MOVL C04706 V=8.0
MOVL C04707 V=8.0
MOVL C04708 V=8.0
MOVL C04709 V=8.0
MOVL C04710 V=8.0
MOVL C04711 V=8.0
MOVL C04712 V=8.0
MOVL C04713 V=8.0
MOVL C04714 V=8.0
MOVL C04715 V=8.0
MOVL C04716 V=8.0
MOVL C04717 V=8.0
MOVL C04718 V=8.0
MOVL C04719 V=8.0
MOVL C04720 V=8.0
MOVL C04721 V=8.0
MOVL C04722 V=8.0
MOVJ C04723 VJ=0.78
MOVJ C04724 VJ=0.78
MOVL C04725 V=11.7
TIMER T=2.00
MOVL C04726 V=11.7
MOVJ C04727 VJ=0.78
MOVJ C04728 VJ=0.78
MOVL C04729 V=8.0
MOVL C04730 V=8.0
MOVJ C04731 VJ=0.78
MOVL C04732 V=8.0
MOVL C04733 V=8.0
MOVL C04734 V=8.0
MOVL C04735 V=8.0
MOVL C04736 V=8.0
MOVL C04737 V=8.0
MOVL C04738 V=8.0
MOVL C04739 V=8.0
MOVL C04740 V=8.0
MOVL C04741 V=8.0
MOVL C04742 V=8.0
MOVL C04743 V=8.0
MOVL C04744 V=8.0
MOVL C04745 V=8.0
MOVL C04746 V=8.0
MOVL C04747 V=8.0
MOVL C04748 V=8.0
MOVL C04749 V=8.0
MOVL C04750 V=8.0
MOVL C04751 V=8.0
MOVL C04752 V=8.0
MOVL C04753 V=8.0
MOVL C04754 V=8.0
MOVL C04755 V=8.0
MOVL C04756 V=8.0
MOVL C04757 V=8.0
MOVL C04758 V=8.0
MOVL C04759 V=8.0
MOVL C04760 V=8.0
MOVL C04761 V=8.0
MOVL C04762 V=8.0
MOVL C04763 V=8.0
MOVL C04764 V=8.0
MOVL C04765 V=8.0
MOVL C04766 V=8.0
MOVL C04767 V=8.0
MOVL C04768 V=8.0
MOVL C04769 V=8.0
MOVL C04770 V=8.0
MOVL C04771 V=8.0
MOVL C04772 V=8.0
MOVL C04773 V=8.0
MOVL C04774 V=8.0
MOVL C04775 V=8.0
MOVL C04776 V=8.0
MOVL C04777 V=8.0
MOVL C04778 V=8.0
MOVL C04779 V=8.0
MOVL C04780 V=8.0
MOVL C04781 V=8.0
MOVL C04782 V=8.0
MOVL C04783 V=8.0
MOVL C04784 V=8.0
MOVL C04785 V=8.0
MOVL C04786 V=8.0
MOVL C04787 V=8.0
MOVL C04788 V=8.0
MOVL C04789 V=8.0
MOVL C04790 V=8.0
MOVL C04791 V=8.0
MOVL C04792 V=8.0
MOVL C04793 V=8.0
MOVJ C04794 VJ=0.78
MOVL C04795 V=8.0
MOVL C04796 V=8.0
MOVL C04797 V=8.0
MOVL C04798 V=8.0
MOVL C04799 V=8.0
MOVL C04800 V=8.0
MOVL C04801 V=8.0
MOVL C04802 V=8.0
MOVL C04803 V=8.0
MOVL C04804 V=8.0
MOVL C04805 V=8.0
MOVL C04806 V=8.0
MOVL C04807 V=8.0
MOVL C04808 V=8.0
MOVL C04809 V=8.0
MOVL C04810 V=8.0
MOVL C04811 V=8.0
MOVL C04812 V=8.0
MOVL C04813 V=8.0
MOVL C04814 V=8.0
MOVL C04815 V=8.0
MOVL C04816 V=8.0
MOVL C04817 V=8.0
MOVL C04818 V=8.0
MOVL C04819 V=8.0
MOVL C04820 V=8.0
MOVL C04821 V=8.0
MOVL C04822 V=8.0
MOVL C04823 V=8.0
MOVL C04824 V=8.0
MOVL C04825 V=8.0
MOVL C04826 V=8.0
MOVL C04827 V=8.0
MOVL C04828 V=8.0
MOVL C04829 V=8.0
MOVL C04830 V=8.0
MOVL C04831 V=8.0
MOVL C04832 V=8.0
MOVL C04833 V=8.0
MOVL C04834 V=8.0
MOVL C04835 V=8.0
MOVL C04836 V=8.0
MOVL C04837 V=8.0
MOVL C04838 V=8.0
MOVL C04839 V=8.0
MOVL C04840 V=8.0
MOVL C04841 V=8.0
MOVL C04842 V=8.0
MOVL C04843 V=8.0
MOVL C04844 V=8.0
MOVL C04845 V=8.0
MOVL C04846 V=8.0
MOVL C04847 V=8.0
MOVL C04848 V=8.0
MOVL C04849 V=8.0
MOVL C04850 V=8.0
MOVL C04851 V=8.0
MOVL C04852 V=8.0
MOVL C04853 V=8.0
MOVL C04854 V=8.0
MOVL C04855 V=8.0
MOVL C04856 V=8.0
MOVJ C04857 VJ=0.78
MOVL C04858 V=8.0
MOVL C04859 V=8.0
MOVL C04860 V=8.0
MOVL C04861 V=8.0
MOVL C04862 V=8.0
MOVL C04863 V=8.0
MOVL C04864 V=8.0
MOVL C04865 V=8.0
MOVL C04866 V=8.0
MOVL C04867 V=8.0
MOVL C04868 V=8.0
MOVL C04869 V=8.0
MOVL C04870 V=8.0
MOVL C04871 V=8.0
MOVL C04872 V=8.0
MOVL C04873 V=8.0
MOVL C04874 V=8.0
MOVL C04875 V=8.0
MOVL C04876 V=8.0
MOVL C04877 V=8.0
MOVL C04878 V=8.0
MOVL C04879 V=8.0
MOVL C04880 V=8.0
MOVL C04881 V=8.0
MOVL C04882 V=8.0
MOVL C04883 V=8.0
MOVL C04884 V=8.0
MOVL C04885 V=8.0
MOVL C04886 V=8.0
MOVL C04887 V=8.0
MOVL C04888 V=8.0
MOVL C04889 V=8.0
MOVL C04890 V=8.0
MOVL C04891 V=8.0
MOVL C04892 V=8.0
MOVL C04893 V=8.0
MOVL C04894 V=8.0
MOVL C04895 V=8.0
MOVL C04896 V=8.0
MOVL C04897 V=8.0
MOVL C04898 V=8.0
MOVJ C04899 VJ=0.78
MOVJ C04900 VJ=0.78
MOVL C04901 V=11.7
TIMER T=2.00
MOVL C04902 V=11.7
MOVJ C04903 VJ=0.78
MOVJ C04904 VJ=0.78
MOVL C04905 V=8.0
MOVL C04906 V=8.0
MOVL C04907 V=8.0
MOVL C04908 V=8.0
MOVL C04909 V=8.0
MOVL C04910 V=8.0
MOVL C04911 V=8.0
MOVL C04912 V=8.0
MOVL C04913 V=8.0
MOVL C04914 V=8.0
MOVL C04915 V=8.0
MOVL C04916 V=8.0
MOVL C04917 V=8.0
MOVL C04918 V=8.0
MOVL C04919 V=8.0
MOVL C04920 V=8.0
MOVL C04921 V=8.0
MOVL C04922 V=8.0
MOVL C04923 V=8.0
MOVL C04924 V=8.0
MOVL C04925 V=8.0
MOVL C04926 V=8.0
MOVJ C04927 VJ=0.78
MOVL C04928 V=8.0
MOVL C04929 V=8.0
MOVL C04930 V=8.0
MOVL C04931 V=8.0
MOVL C04932 V=8.0
MOVL C04933 V=8.0
MOVL C04934 V=8.0
MOVL C04935 V=8.0
MOVL C04936 V=8.0
MOVL C04937 V=8.0
MOVL C04938 V=8.0
MOVL C04939 V=8.0
MOVL C04940 V=8.0
MOVL C04941 V=8.0
MOVL C04942 V=8.0
MOVL C04943 V=8.0
MOVL C04944 V=8.0
MOVL C04945 V=8.0
MOVL C04946 V=8.0
MOVL C04947 V=8.0
MOVL C04948 V=8.0
MOVL C04949 V=8.0
MOVL C04950 V=8.0
MOVL C04951 V=8.0
MOVL C04952 V=8.0
MOVL C04953 V=8.0
MOVL C04954 V=8.0
MOVL C04955 V=8.0
MOVL C04956 V=8.0
MOVL C04957 V=8.0
MOVL C04958 V=8.0
MOVL C04959 V=8.0
MOVL C04960 V=8.0
MOVL C04961 V=8.0
MOVL C04962 V=8.0
MOVL C04963 V=8.0
MOVL C04964 V=8.0
MOVL C04965 V=8.0
MOVL C04966 V=8.0
MOVL C04967 V=8.0
MOVL C04968 V=8.0
MOVL C04969 V=8.0
MOVL C04970 V=8.0
MOVL C04971 V=8.0
MOVL C04972 V=8.0
MOVL C04973 V=8.0
MOVL C04974 V=8.0
MOVL C04975 V=8.0
MOVL C04976 V=8.0
MOVL C04977 V=8.0
MOVL C04978 V=8.0
MOVL C04979 V=8.0
MOVL C04980 V=8.0
MOVL C04981 V=8.0
MOVL C04982 V=8.0
MOVL C04983 V=8.0
MOVL C04984 V=8.0
MOVL C04985 V=8.0
MOVL C04986 V=8.0
MOVL C04987 V=8.0
MOVL C04988 V=8.0
MOVL C04989 V=8.0
MOVJ C04990 VJ=0.78
MOVL C04991 V=8.0
MOVL C04992 V=8.0
MOVL C04993 V=8.0
MOVL C04994 V=8.0
MOVL C04995 V=8.0
MOVL C04996 V=8.0
MOVL C04997 V=8.0
MOVL C04998 V=8.0
MOVL C04999 V=8.0
MOVL C05000 V=8.0
MOVL C05001 V=8.0
MOVL C05002 V=8.0
MOVL C05003 V=8.0
MOVL C05004 V=8.0
MOVL C05005 V=8.0
MOVL C05006 V=8.0
MOVL C05007 V=8.0
MOVL C05008 V=8.0
MOVL C05009 V=8.0
MOVL C05010 V=8.0
MOVL C05011 V=8.0
MOVL C05012 V=8.0
MOVL C05013 V=8.0
MOVL C05014 V=8.0
MOVL C05015 V=8.0
MOVL C05016 V=8.0
MOVL C05017 V=8.0
MOVL C05018 V=8.0
MOVL C05019 V=8.0
MOVL C05020 V=8.0
MOVL C05021 V=8.0
MOVL C05022 V=8.0
MOVL C05023 V=8.0
MOVL C05024 V=8.0
MOVL C05025 V=8.0
MOVL C05026 V=8.0
MOVL C05027 V=8.0
MOVL C05028 V=8.0
MOVL C05029 V=8.0
MOVL C05030 V=8.0
MOVL C05031 V=8.0
MOVL C05032 V=8.0
MOVL C05033 V=8.0
MOVL C05034 V=8.0
MOVL C05035 V=8.0
MOVL C05036 V=8.0
MOVL C05037 V=8.0
MOVL C05038 V=8.0
MOVL C05039 V=8.0
MOVL C05040 V=8.0
MOVL C05041 V=8.0
MOVL C05042 V=8.0
MOVL C05043 V=8.0
MOVL C05044 V=8.0
MOVL C05045 V=8.0
MOVL C05046 V=8.0
MOVL C05047 V=8.0
MOVL C05048 V=8.0
MOVL C05049 V=8.0
MOVL C05050 V=8.0
MOVL C05051 V=8.0
MOVL C05052 V=8.0
MOVJ C05053 VJ=0.78
MOVL C05054 V=8.0
MOVL C05055 V=8.0
MOVL C05056 V=8.0
MOVL C05057 V=8.0
MOVL C05058 V=8.0
MOVL C05059 V=8.0
MOVL C05060 V=8.0
MOVL C05061 V=8.0
MOVL C05062 V=8.0
MOVL C05063 V=8.0
MOVL C05064 V=8.0
MOVL C05065 V=8.0
MOVL C05066 V=8.0
MOVL C05067 V=8.0
MOVL C05068 V=8.0
MOVL C05069 V=8.0
MOVL C05070 V=8.0
MOVL C05071 V=8.0
MOVL C05072 V=8.0
MOVL C05073 V=8.0
MOVL C05074 V=8.0
MOVJ C05075 VJ=0.78
MOVJ C05076 VJ=0.78
MOVL C05077 V=11.7
TIMER T=2.00
MOVL C05078 V=11.7
MOVJ C05079 VJ=0.78
MOVJ C05080 VJ=0.78
MOVL C05081 V=8.0
MOVL C05082 V=8.0
MOVL C05083 V=8.0
MOVL C05084 V=8.0
MOVL C05085 V=8.0
MOVL C05086 V=8.0
MOVL C05087 V=8.0
MOVL C05088 V=8.0
MOVL C05089 V=8.0
MOVL C05090 V=8.0
MOVL C05091 V=8.0
MOVL C05092 V=8.0
MOVL C05093 V=8.0
MOVL C05094 V=8.0
MOVL C05095 V=8.0
MOVL C05096 V=8.0
MOVL C05097 V=8.0
MOVL C05098 V=8.0
MOVL C05099 V=8.0
MOVL C05100 V=8.0
MOVL C05101 V=8.0
MOVL C05102 V=8.0
MOVL C05103 V=8.0
MOVL C05104 V=8.0
MOVL C05105 V=8.0
MOVL C05106 V=8.0
MOVL C05107 V=8.0
MOVL C05108 V=8.0
MOVL C05109 V=8.0
MOVL C05110 V=8.0
MOVL C05111 V=8.0
MOVL C05112 V=8.0
MOVL C05113 V=8.0
MOVL C05114 V=8.0
MOVL C05115 V=8.0
MOVL C05116 V=8.0
MOVL C05117 V=8.0
MOVL C05118 V=8.0
MOVL C05119 V=8.0
MOVL C05120 V=8.0
MOVL C05121 V=8.0
MOVL C05122 V=8.0
MOVJ C05123 VJ=0.78
MOVL C05124 V=8.0
MOVL C05125 V=8.0
MOVL C05126 V=8.0
MOVL C05127 V=8.0
MOVL C05128 V=8.0
MOVL C05129 V=8.0
MOVL C05130 V=8.0
MOVL C05131 V=8.0
MOVL C05132 V=8.0
MOVL C05133 V=8.0
MOVL C05134 V=8.0
MOVL C05135 V=8.0
MOVL C05136 V=8.0
MOVL C05137 V=8.0
MOVL C05138 V=8.0
MOVL C05139 V=8.0
MOVL C05140 V=8.0
MOVL C05141 V=8.0
MOVL C05142 V=8.0
MOVL C05143 V=8.0
MOVL C05144 V=8.0
MOVL C05145 V=8.0
MOVL C05146 V=8.0
MOVL C05147 V=8.0
MOVL C05148 V=8.0
MOVL C05149 V=8.0
MOVL C05150 V=8.0
MOVL C05151 V=8.0
MOVL C05152 V=8.0
MOVL C05153 V=8.0
MOVL C05154 V=8.0
MOVL C05155 V=8.0
MOVL C05156 V=8.0
MOVL C05157 V=8.0
MOVL C05158 V=8.0
MOVL C05159 V=8.0
MOVL C05160 V=8.0
MOVL C05161 V=8.0
MOVL C05162 V=8.0
MOVL C05163 V=8.0
MOVL C05164 V=8.0
MOVL C05165 V=8.0
MOVL C05166 V=8.0
MOVL C05167 V=8.0
MOVL C05168 V=8.0
MOVL C05169 V=8.0
MOVL C05170 V=8.0
MOVL C05171 V=8.0
MOVL C05172 V=8.0
MOVL C05173 V=8.0
MOVL C05174 V=8.0
MOVL C05175 V=8.0
MOVL C05176 V=8.0
MOVL C05177 V=8.0
MOVL C05178 V=8.0
MOVL C05179 V=8.0
MOVL C05180 V=8.0
MOVL C05181 V=8.0
MOVL C05182 V=8.0
MOVL C05183 V=8.0
MOVL C05184 V=8.0
MOVL C05185 V=8.0
MOVJ C05186 VJ=0.78
MOVL C05187 V=8.0
MOVL C05188 V=8.0
MOVL C05189 V=8.0
MOVL C05190 V=8.0
MOVL C05191 V=8.0
MOVL C05192 V=8.0
MOVL C05193 V=8.0
MOVL C05194 V=8.0
MOVL C05195 V=8.0
MOVL C05196 V=8.0
MOVL C05197 V=8.0
MOVL C05198 V=8.0
MOVL C05199 V=8.0
MOVL C05200 V=8.0
MOVL C05201 V=8.0
MOVL C05202 V=8.0
MOVL C05203 V=8.0
MOVL C05204 V=8.0
MOVL C05205 V=8.0
MOVL C05206 V=8.0
MOVL C05207 V=8.0
MOVL C05208 V=8.0
MOVL C05209 V=8.0
MOVL C05210 V=8.0
MOVL C05211 V=8.0
MOVL C05212 V=8.0
MOVL C05213 V=8.0
MOVL C05214 V=8.0
MOVL C05215 V=8.0
MOVL C05216 V=8.0
MOVL C05217 V=8.0
MOVL C05218 V=8.0
MOVL C05219 V=8.0
MOVL C05220 V=8.0
MOVL C05221 V=8.0
MOVL C05222 V=8.0
MOVL C05223 V=8.0
MOVL C05224 V=8.0
MOVL C05225 V=8.0
MOVL C05226 V=8.0
MOVL C05227 V=8.0
MOVL C05228 V=8.0
MOVL C05229 V=8.0
MOVL C05230 V=8.0
MOVL C05231 V=8.0
MOVL C05232 V=8.0
MOVL C05233 V=8.0
MOVL C05234 V=8.0
MOVL C05235 V=8.0
MOVL C05236 V=8.0
MOVL C05237 V=8.0
MOVL C05238 V=8.0
MOVL C05239 V=8.0
MOVL C05240 V=8.0
MOVL C05241 V=8.0
MOVL C05242 V=8.0
MOVL C05243 V=8.0
MOVL C05244 V=8.0
MOVL C05245 V=8.0
MOVL C05246 V=8.0
MOVL C05247 V=8.0
MOVJ C05248 VJ=0.78
MOVJ C05249 VJ=0.78
MOVL C05250 V=11.7
TIMER T=2.00
MOVL C05251 V=11.7
MOVJ C05252 VJ=0.78
MOVJ C05253 VJ=0.78
MOVL C05254 V=8.0
MOVL C05255 V=8.0
MOVJ C05256 VJ=0.78
MOVL C05257 V=8.0
MOVL C05258 V=8.0
MOVL C05259 V=8.0
MOVL C05260 V=8.0
MOVL C05261 V=8.0
MOVL C05262 V=8.0
MOVL C05263 V=8.0
MOVL C05264 V=8.0
MOVL C05265 V=8.0
MOVL C05266 V=8.0
MOVL C05267 V=8.0
MOVL C05268 V=8.0
MOVL C05269 V=8.0
MOVL C05270 V=8.0
MOVL C05271 V=8.0
MOVL C05272 V=8.0
MOVL C05273 V=8.0
MOVL C05274 V=8.0
MOVL C05275 V=8.0
MOVL C05276 V=8.0
MOVL C05277 V=8.0
MOVL C05278 V=8.0
MOVL C05279 V=8.0
MOVL C05280 V=8.0
MOVL C05281 V=8.0
MOVL C05282 V=8.0
MOVL C05283 V=8.0
MOVL C05284 V=8.0
MOVL C05285 V=8.0
MOVL C05286 V=8.0
MOVL C05287 V=8.0
MOVL C05288 V=8.0
MOVL C05289 V=8.0
MOVL C05290 V=8.0
MOVL C05291 V=8.0
MOVL C05292 V=8.0
MOVL C05293 V=8.0
MOVL C05294 V=8.0
MOVL C05295 V=8.0
MOVL C05296 V=8.0
MOVL C05297 V=8.0
MOVL C05298 V=8.0
MOVL C05299 V=8.0
MOVL C05300 V=8.0
MOVL C05301 V=8.0
MOVL C05302 V=8.0
MOVL C05303 V=8.0
MOVL C05304 V=8.0
MOVL C05305 V=8.0
MOVL C05306 V=8.0
MOVL C05307 V=8.0
MOVL C05308 V=8.0
MOVL C05309 V=8.0
MOVL C05310 V=8.0
MOVL C05311 V=8.0
MOVL C05312 V=8.0
MOVL C05313 V=8.0
MOVL C05314 V=8.0
MOVL C05315 V=8.0
MOVL C05316 V=8.0
MOVL C05317 V=8.0
MOVL C05318 V=8.0
MOVJ C05319 VJ=0.78
MOVL C05320 V=8.0
MOVL C05321 V=8.0
MOVL C05322 V=8.0
MOVL C05323 V=8.0
MOVL C05324 V=8.0
MOVL C05325 V=8.0
MOVL C05326 V=8.0
MOVL C05327 V=8.0
MOVL C05328 V=8.0
MOVL C05329 V=8.0
MOVL C05330 V=8.0
MOVL C05331 V=8.0
MOVL C05332 V=8.0
MOVL C05333 V=8.0
MOVL C05334 V=8.0
MOVL C05335 V=8.0
MOVL C05336 V=8.0
MOVL C05337 V=8.0
MOVL C05338 V=8.0
MOVL C05339 V=8.0
MOVL C05340 V=8.0
MOVL C05341 V=8.0
MOVL C05342 V=8.0
MOVL C05343 V=8.0
MOVL C05344 V=8.0
MOVL C05345 V=8.0
MOVL C05346 V=8.0
MOVL C05347 V=8.0
MOVL C05348 V=8.0
MOVL C05349 V=8.0
MOVL C05350 V=8.0
MOVL C05351 V=8.0
MOVL C05352 V=8.0
MOVL C05353 V=8.0
MOVL C05354 V=8.0
MOVL C05355 V=8.0
MOVL C05356 V=8.0
MOVL C05357 V=8.0
MOVL C05358 V=8.0
MOVL C05359 V=8.0
MOVL C05360 V=8.0
MOVL C05361 V=8.0
MOVL C05362 V=8.0
MOVL C05363 V=8.0
MOVL C05364 V=8.0
MOVL C05365 V=8.0
MOVL C05366 V=8.0
MOVL C05367 V=8.0
MOVL C05368 V=8.0
MOVL C05369 V=8.0
MOVL C05370 V=8.0
MOVL C05371 V=8.0
MOVL C05372 V=8.0
MOVL C05373 V=8.0
MOVL C05374 V=8.0
MOVL C05375 V=8.0
MOVL C05376 V=8.0
MOVL C05377 V=8.0
MOVL C05378 V=8.0
MOVL C05379 V=8.0
MOVL C05380 V=8.0
MOVL C05381 V=8.0
MOVJ C05382 VJ=0.78
MOVL C05383 V=8.0
MOVL C05384 V=8.0
MOVL C05385 V=8.0
MOVL C05386 V=8.0
MOVL C05387 V=8.0
MOVL C05388 V=8.0
MOVL C05389 V=8.0
MOVL C05390 V=8.0
MOVL C05391 V=8.0
MOVL C05392 V=8.0
MOVL C05393 V=8.0
MOVL C05394 V=8.0
MOVL C05395 V=8.0
MOVL C05396 V=8.0
MOVL C05397 V=8.0
MOVL C05398 V=8.0
MOVL C05399 V=8.0
MOVL C05400 V=8.0
MOVL C05401 V=8.0
MOVL C05402 V=8.0
MOVL C05403 V=8.0
MOVL C05404 V=8.0
MOVL C05405 V=8.0
MOVL C05406 V=8.0
MOVL C05407 V=8.0
MOVL C05408 V=8.0
MOVL C05409 V=8.0
MOVL C05410 V=8.0
MOVL C05411 V=8.0
MOVL C05412 V=8.0
MOVL C05413 V=8.0
MOVL C05414 V=8.0
MOVL C05415 V=8.0
MOVL C05416 V=8.0
MOVL C05417 V=8.0
MOVL C05418 V=8.0
MOVL C05419 V=8.0
MOVL C05420 V=8.0
MOVL C05421 V=8.0
MOVL C05422 V=8.0
MOVL C05423 V=8.0
MOVJ C05424 VJ=0.78
MOVJ C05425 VJ=0.78
MOVL C05426 V=11.7
TIMER T=2.00
MOVL C05427 V=11.7
MOVJ C05428 VJ=0.78
MOVJ C05429 VJ=0.78
MOVL C05430 V=8.0
MOVL C05431 V=8.0
MOVL C05432 V=8.0
MOVL C05433 V=8.0
MOVL C05434 V=8.0
MOVL C05435 V=8.0
MOVL C05436 V=8.0
MOVL C05437 V=8.0
MOVL C05438 V=8.0
MOVL C05439 V=8.0
MOVL C05440 V=8.0
MOVL C05441 V=8.0
MOVL C05442 V=8.0
MOVL C05443 V=8.0
MOVL C05444 V=8.0
MOVL C05445 V=8.0
MOVL C05446 V=8.0
MOVL C05447 V=8.0
MOVL C05448 V=8.0
MOVL C05449 V=8.0
MOVL C05450 V=8.0
MOVL C05451 V=8.0
MOVJ C05452 VJ=0.78
MOVL C05453 V=8.0
MOVL C05454 V=8.0
MOVL C05455 V=8.0
MOVL C05456 V=8.0
MOVL C05457 V=8.0
MOVL C05458 V=8.0
MOVL C05459 V=8.0
MOVL C05460 V=8.0
MOVL C05461 V=8.0
MOVL C05462 V=8.0
MOVL C05463 V=8.0
MOVL C05464 V=8.0
MOVL C05465 V=8.0
MOVL C05466 V=8.0
MOVL C05467 V=8.0
MOVL C05468 V=8.0
MOVL C05469 V=8.0
MOVL C05470 V=8.0
MOVL C05471 V=8.0
MOVL C05472 V=8.0
MOVL C05473 V=8.0
MOVL C05474 V=8.0
MOVL C05475 V=8.0
MOVL C05476 V=8.0
MOVL C05477 V=8.0
MOVL C05478 V=8.0
MOVL C05479 V=8.0
MOVL C05480 V=8.0
MOVL C05481 V=8.0
MOVL C05482 V=8.0
MOVL C05483 V=8.0
MOVL C05484 V=8.0
MOVL C05485 V=8.0
MOVL C05486 V=8.0
MOVL C05487 V=8.0
MOVL C05488 V=8.0
MOVL C05489 V=8.0
MOVL C05490 V=8.0
MOVL C05491 V=8.0
MOVL C05492 V=8.0
MOVL C05493 V=8.0
MOVL C05494 V=8.0
MOVL C05495 V=8.0
MOVL C05496 V=8.0
MOVL C05497 V=8.0
MOVL C05498 V=8.0
MOVL C05499 V=8.0
MOVL C05500 V=8.0
MOVL C05501 V=8.0
MOVL C05502 V=8.0
MOVL C05503 V=8.0
MOVL C05504 V=8.0
MOVL C05505 V=8.0
MOVL C05506 V=8.0
MOVL C05507 V=8.0
MOVL C05508 V=8.0
MOVL C05509 V=8.0
MOVL C05510 V=8.0
MOVL C05511 V=8.0
MOVL C05512 V=8.0
MOVL C05513 V=8.0
MOVL C05514 V=8.0
MOVJ C05515 VJ=0.78
MOVL C05516 V=8.0
MOVL C05517 V=8.0
MOVL C05518 V=8.0
MOVL C05519 V=8.0
MOVL C05520 V=8.0
MOVL C05521 V=8.0
MOVL C05522 V=8.0
MOVL C05523 V=8.0
MOVL C05524 V=8.0
MOVL C05525 V=8.0
MOVL C05526 V=8.0
MOVL C05527 V=8.0
MOVL C05528 V=8.0
MOVL C05529 V=8.0
MOVL C05530 V=8.0
MOVL C05531 V=8.0
MOVL C05532 V=8.0
MOVL C05533 V=8.0
MOVL C05534 V=8.0
MOVL C05535 V=8.0
MOVL C05536 V=8.0
MOVL C05537 V=8.0
MOVL C05538 V=8.0
MOVL C05539 V=8.0
MOVL C05540 V=8.0
MOVL C05541 V=8.0
MOVL C05542 V=8.0
MOVL C05543 V=8.0
MOVL C05544 V=8.0
MOVL C05545 V=8.0
MOVL C05546 V=8.0
MOVL C05547 V=8.0
MOVL C05548 V=8.0
MOVL C05549 V=8.0
MOVL C05550 V=8.0
MOVL C05551 V=8.0
MOVL C05552 V=8.0
MOVL C05553 V=8.0
MOVL C05554 V=8.0
MOVL C05555 V=8.0
MOVL C05556 V=8.0
MOVL C05557 V=8.0
MOVL C05558 V=8.0
MOVL C05559 V=8.0
MOVL C05560 V=8.0
MOVL C05561 V=8.0
MOVL C05562 V=8.0
MOVL C05563 V=8.0
MOVL C05564 V=8.0
MOVL C05565 V=8.0
MOVL C05566 V=8.0
MOVL C05567 V=8.0
MOVL C05568 V=8.0
MOVL C05569 V=8.0
MOVL C05570 V=8.0
MOVL C05571 V=8.0
MOVL C05572 V=8.0
MOVL C05573 V=8.0
MOVL C05574 V=8.0
MOVL C05575 V=8.0
MOVL C05576 V=8.0
MOVL C05577 V=8.0
MOVJ C05578 VJ=0.78
MOVL C05579 V=8.0
MOVL C05580 V=8.0
MOVL C05581 V=8.0
MOVL C05582 V=8.0
MOVL C05583 V=8.0
MOVL C05584 V=8.0
MOVL C05585 V=8.0
MOVL C05586 V=8.0
MOVL C05587 V=8.0
MOVL C05588 V=8.0
MOVL C05589 V=8.0
MOVL C05590 V=8.0
MOVL C05591 V=8.0
MOVL C05592 V=8.0
MOVL C05593 V=8.0
MOVL C05594 V=8.0
MOVL C05595 V=8.0
MOVL C05596 V=8.0
MOVL C05597 V=8.0
MOVL C05598 V=8.0
MOVL C05599 V=8.0
MOVJ C05600 VJ=0.78
MOVJ C05601 VJ=0.78
MOVL C05602 V=11.7
TIMER T=2.00
MOVL C05603 V=11.7
MOVJ C05604 VJ=0.78
MOVJ C05605 VJ=0.78
MOVL C05606 V=8.0
MOVL C05607 V=8.0
MOVL C05608 V=8.0
MOVL C05609 V=8.0
MOVL C05610 V=8.0
MOVL C05611 V=8.0
MOVL C05612 V=8.0
MOVL C05613 V=8.0
MOVL C05614 V=8.0
MOVL C05615 V=8.0
MOVL C05616 V=8.0
MOVL C05617 V=8.0
MOVL C05618 V=8.0
MOVL C05619 V=8.0
MOVL C05620 V=8.0
MOVL C05621 V=8.0
MOVL C05622 V=8.0
MOVL C05623 V=8.0
MOVL C05624 V=8.0
MOVL C05625 V=8.0
MOVL C05626 V=8.0
MOVL C05627 V=8.0
MOVL C05628 V=8.0
MOVL C05629 V=8.0
MOVL C05630 V=8.0
MOVL C05631 V=8.0
MOVL C05632 V=8.0
MOVL C05633 V=8.0
MOVL C05634 V=8.0
MOVL C05635 V=8.0
MOVL C05636 V=8.0
MOVL C05637 V=8.0
MOVL C05638 V=8.0
MOVL C05639 V=8.0
MOVL C05640 V=8.0
MOVL C05641 V=8.0
MOVL C05642 V=8.0
MOVL C05643 V=8.0
MOVL C05644 V=8.0
MOVL C05645 V=8.0
MOVL C05646 V=8.0
MOVL C05647 V=8.0
MOVJ C05648 VJ=0.78
MOVL C05649 V=8.0
MOVL C05650 V=8.0
MOVL C05651 V=8.0
MOVL C05652 V=8.0
MOVL C05653 V=8.0
MOVL C05654 V=8.0
MOVL C05655 V=8.0
MOVL C05656 V=8.0
MOVL C05657 V=8.0
MOVL C05658 V=8.0
MOVL C05659 V=8.0
MOVL C05660 V=8.0
MOVL C05661 V=8.0
MOVL C05662 V=8.0
MOVL C05663 V=8.0
MOVL C05664 V=8.0
MOVL C05665 V=8.0
MOVL C05666 V=8.0
MOVL C05667 V=8.0
MOVL C05668 V=8.0
MOVL C05669 V=8.0
MOVL C05670 V=8.0
MOVL C05671 V=8.0
MOVL C05672 V=8.0
MOVL C05673 V=8.0
MOVL C05674 V=8.0
MOVL C05675 V=8.0
MOVL C05676 V=8.0
MOVL C05677 V=8.0
MOVL C05678 V=8.0
MOVL C05679 V=8.0
MOVL C05680 V=8.0
MOVL C05681 V=8.0
MOVL C05682 V=8.0
MOVL C05683 V=8.0
MOVL C05684 V=8.0
MOVL C05685 V=8.0
MOVL C05686 V=8.0
MOVL C05687 V=8.0
MOVL C05688 V=8.0
MOVL C05689 V=8.0
MOVL C05690 V=8.0
MOVL C05691 V=8.0
MOVL C05692 V=8.0
MOVL C05693 V=8.0
MOVL C05694 V=8.0
MOVL C05695 V=8.0
MOVL C05696 V=8.0
MOVL C05697 V=8.0
MOVL C05698 V=8.0
MOVL C05699 V=8.0
MOVL C05700 V=8.0
MOVL C05701 V=8.0
MOVL C05702 V=8.0
MOVL C05703 V=8.0
MOVL C05704 V=8.0
MOVL C05705 V=8.0
MOVL C05706 V=8.0
MOVL C05707 V=8.0
MOVL C05708 V=8.0
MOVL C05709 V=8.0
MOVL C05710 V=8.0
MOVJ C05711 VJ=0.78
MOVL C05712 V=8.0
MOVL C05713 V=8.0
MOVL C05714 V=8.0
MOVL C05715 V=8.0
MOVL C05716 V=8.0
MOVL C05717 V=8.0
MOVL C05718 V=8.0
MOVL C05719 V=8.0
MOVL C05720 V=8.0
MOVL C05721 V=8.0
MOVL C05722 V=8.0
MOVL C05723 V=8.0
MOVL C05724 V=8.0
MOVL C05725 V=8.0
MOVL C05726 V=8.0
MOVL C05727 V=8.0
MOVL C05728 V=8.0
MOVL C05729 V=8.0
MOVL C05730 V=8.0
MOVL C05731 V=8.0
MOVL C05732 V=8.0
MOVL C05733 V=8.0
MOVL C05734 V=8.0
MOVL C05735 V=8.0
MOVL C05736 V=8.0
MOVL C05737 V=8.0
MOVL C05738 V=8.0
MOVL C05739 V=8.0
MOVL C05740 V=8.0
MOVL C05741 V=8.0
MOVL C05742 V=8.0
MOVL C05743 V=8.0
MOVL C05744 V=8.0
MOVL C05745 V=8.0
MOVL C05746 V=8.0
MOVL C05747 V=8.0
MOVL C05748 V=8.0
MOVL C05749 V=8.0
MOVL C05750 V=8.0
MOVL C05751 V=8.0
MOVL C05752 V=8.0
MOVL C05753 V=8.0
MOVL C05754 V=8.0
MOVL C05755 V=8.0
MOVL C05756 V=8.0
MOVL C05757 V=8.0
MOVL C05758 V=8.0
MOVL C05759 V=8.0
MOVL C05760 V=8.0
MOVL C05761 V=8.0
MOVL C05762 V=8.0
MOVL C05763 V=8.0
MOVL C05764 V=8.0
MOVL C05765 V=8.0
MOVL C05766 V=8.0
MOVL C05767 V=8.0
MOVL C05768 V=8.0
MOVL C05769 V=8.0
MOVL C05770 V=8.0
MOVL C05771 V=8.0
MOVL C05772 V=8.0
MOVJ C05773 VJ=0.78
MOVJ C05774 VJ=0.78
MOVL C05775 V=11.7
TIMER T=2.00
MOVL C05776 V=11.7
MOVJ C05777 VJ=0.78
MOVJ C05778 VJ=0.78
MOVL C05779 V=8.0
MOVL C05780 V=8.0
MOVJ C05781 VJ=0.78
MOVL C05782 V=8.0
MOVL C05783 V=8.0
MOVL C05784 V=8.0
MOVL C05785 V=8.0
MOVL C05786 V=8.0
MOVL C05787 V=8.0
MOVL C05788 V=8.0
MOVL C05789 V=8.0
MOVL C05790 V=8.0
MOVL C05791 V=8.0
MOVL C05792 V=8.0
MOVL C05793 V=8.0
MOVL C05794 V=8.0
MOVL C05795 V=8.0
MOVL C05796 V=8.0
MOVL C05797 V=8.0
MOVL C05798 V=8.0
MOVL C05799 V=8.0
MOVL C05800 V=8.0
MOVL C05801 V=8.0
MOVL C05802 V=8.0
MOVL C05803 V=8.0
MOVL C05804 V=8.0
MOVL C05805 V=8.0
MOVL C05806 V=8.0
MOVL C05807 V=8.0
MOVL C05808 V=8.0
MOVL C05809 V=8.0
MOVL C05810 V=8.0
MOVL C05811 V=8.0
MOVL C05812 V=8.0
MOVL C05813 V=8.0
MOVL C05814 V=8.0
MOVL C05815 V=8.0
MOVL C05816 V=8.0
MOVL C05817 V=8.0
MOVL C05818 V=8.0
MOVL C05819 V=8.0
MOVL C05820 V=8.0
MOVL C05821 V=8.0
MOVL C05822 V=8.0
MOVL C05823 V=8.0
MOVL C05824 V=8.0
MOVL C05825 V=8.0
MOVL C05826 V=8.0
MOVL C05827 V=8.0
MOVL C05828 V=8.0
MOVL C05829 V=8.0
MOVL C05830 V=8.0
MOVL C05831 V=8.0
MOVL C05832 V=8.0
MOVL C05833 V=8.0
MOVL C05834 V=8.0
MOVL C05835 V=8.0
MOVL C05836 V=8.0
MOVL C05837 V=8.0
MOVL C05838 V=8.0
MOVL C05839 V=8.0
MOVL C05840 V=8.0
MOVL C05841 V=8.0
MOVL C05842 V=8.0
MOVL C05843 V=8.0
MOVJ C05844 VJ=0.78
MOVL C05845 V=8.0
MOVL C05846 V=8.0
MOVL C05847 V=8.0
MOVL C05848 V=8.0
MOVL C05849 V=8.0
MOVL C05850 V=8.0
MOVL C05851 V=8.0
MOVL C05852 V=8.0
MOVL C05853 V=8.0
MOVL C05854 V=8.0
MOVL C05855 V=8.0
MOVL C05856 V=8.0
MOVL C05857 V=8.0
MOVL C05858 V=8.0
MOVL C05859 V=8.0
MOVL C05860 V=8.0
MOVL C05861 V=8.0
MOVL C05862 V=8.0
MOVL C05863 V=8.0
MOVL C05864 V=8.0
MOVL C05865 V=8.0
MOVL C05866 V=8.0
MOVL C05867 V=8.0
MOVL C05868 V=8.0
MOVL C05869 V=8.0
MOVL C05870 V=8.0
MOVL C05871 V=8.0
MOVL C05872 V=8.0
MOVL C05873 V=8.0
MOVL C05874 V=8.0
MOVL C05875 V=8.0
MOVL C05876 V=8.0
MOVL C05877 V=8.0
MOVL C05878 V=8.0
MOVL C05879 V=8.0
MOVL C05880 V=8.0
MOVL C05881 V=8.0
MOVL C05882 V=8.0
MOVL C05883 V=8.0
MOVL C05884 V=8.0
MOVL C05885 V=8.0
MOVL C05886 V=8.0
MOVL C05887 V=8.0
MOVL C05888 V=8.0
MOVL C05889 V=8.0
MOVL C05890 V=8.0
MOVL C05891 V=8.0
MOVL C05892 V=8.0
MOVL C05893 V=8.0
MOVL C05894 V=8.0
MOVL C05895 V=8.0
MOVL C05896 V=8.0
MOVL C05897 V=8.0
MOVL C05898 V=8.0
MOVL C05899 V=8.0
MOVL C05900 V=8.0
MOVL C05901 V=8.0
MOVL C05902 V=8.0
MOVL C05903 V=8.0
MOVL C05904 V=8.0
MOVL C05905 V=8.0
MOVL C05906 V=8.0
MOVJ C05907 VJ=0.78
MOVL C05908 V=8.0
MOVL C05909 V=8.0
MOVL C05910 V=8.0
MOVL C05911 V=8.0
MOVL C05912 V=8.0
MOVL C05913 V=8.0
MOVL C05914 V=8.0
MOVL C05915 V=8.0
MOVL C05916 V=8.0
MOVL C05917 V=8.0
MOVL C05918 V=8.0
MOVL C05919 V=8.0
MOVL C05920 V=8.0
MOVL C05921 V=8.0
MOVL C05922 V=8.0
MOVL C05923 V=8.0
MOVL C05924 V=8.0
MOVL C05925 V=8.0
MOVL C05926 V=8.0
MOVL C05927 V=8.0
MOVL C05928 V=8.0
MOVL C05929 V=8.0
MOVL C05930 V=8.0
MOVL C05931 V=8.0
MOVL C05932 V=8.0
MOVL C05933 V=8.0
MOVL C05934 V=8.0
MOVL C05935 V=8.0
MOVL C05936 V=8.0
MOVL C05937 V=8.0
MOVL C05938 V=8.0
MOVL C05939 V=8.0
MOVL C05940 V=8.0
MOVL C05941 V=8.0
MOVL C05942 V=8.0
MOVL C05943 V=8.0
MOVL C05944 V=8.0
MOVL C05945 V=8.0
MOVL C05946 V=8.0
MOVL C05947 V=8.0
MOVL C05948 V=8.0
MOVJ C05949 VJ=0.78
MOVJ C05950 VJ=0.78
MOVL C05951 V=11.7
TIMER T=2.00
MOVL C05952 V=11.7
MOVJ C05953 VJ=0.78
MOVJ C05954 VJ=0.78
MOVL C05955 V=8.0
MOVL C05956 V=8.0
MOVL C05957 V=8.0
MOVL C05958 V=8.0
MOVL C05959 V=8.0
MOVL C05960 V=8.0
MOVL C05961 V=8.0
MOVL C05962 V=8.0
MOVL C05963 V=8.0
MOVL C05964 V=8.0
MOVL C05965 V=8.0
MOVL C05966 V=8.0
MOVL C05967 V=8.0
MOVL C05968 V=8.0
MOVL C05969 V=8.0
MOVL C05970 V=8.0
MOVL C05971 V=8.0
MOVL C05972 V=8.0
MOVL C05973 V=8.0
MOVL C05974 V=8.0
MOVL C05975 V=8.0
MOVL C05976 V=8.0
MOVJ C05977 VJ=0.78
MOVL C05978 V=8.0
MOVL C05979 V=8.0
MOVL C05980 V=8.0
MOVL C05981 V=8.0
MOVL C05982 V=8.0
MOVL C05983 V=8.0
MOVL C05984 V=8.0
MOVL C05985 V=8.0
MOVL C05986 V=8.0
MOVL C05987 V=8.0
MOVL C05988 V=8.0
MOVL C05989 V=8.0
MOVL C05990 V=8.0
MOVL C05991 V=8.0
MOVL C05992 V=8.0
MOVL C05993 V=8.0
MOVL C05994 V=8.0
MOVL C05995 V=8.0
MOVL C05996 V=8.0
MOVL C05997 V=8.0
MOVL C05998 V=8.0
MOVL C05999 V=8.0
MOVL C06000 V=8.0
MOVL C06001 V=8.0
MOVL C06002 V=8.0
MOVL C06003 V=8.0
MOVL C06004 V=8.0
MOVL C06005 V=8.0
MOVL C06006 V=8.0
MOVL C06007 V=8.0
MOVL C06008 V=8.0
MOVL C06009 V=8.0
MOVL C06010 V=8.0
MOVL C06011 V=8.0
MOVL C06012 V=8.0
MOVL C06013 V=8.0
MOVL C06014 V=8.0
MOVL C06015 V=8.0
MOVL C06016 V=8.0
MOVL C06017 V=8.0
MOVL C06018 V=8.0
MOVL C06019 V=8.0
MOVL C06020 V=8.0
MOVL C06021 V=8.0
MOVL C06022 V=8.0
MOVL C06023 V=8.0
MOVL C06024 V=8.0
MOVL C06025 V=8.0
MOVL C06026 V=8.0
MOVL C06027 V=8.0
MOVL C06028 V=8.0
MOVL C06029 V=8.0
MOVL C06030 V=8.0
MOVL C06031 V=8.0
MOVL C06032 V=8.0
MOVL C06033 V=8.0
MOVL C06034 V=8.0
MOVL C06035 V=8.0
MOVL C06036 V=8.0
MOVL C06037 V=8.0
MOVL C06038 V=8.0
MOVL C06039 V=8.0
MOVJ C06040 VJ=0.78
MOVL C06041 V=8.0
MOVL C06042 V=8.0
MOVL C06043 V=8.0
MOVL C06044 V=8.0
MOVL C06045 V=8.0
MOVL C06046 V=8.0
MOVL C06047 V=8.0
MOVL C06048 V=8.0
MOVL C06049 V=8.0
MOVL C06050 V=8.0
MOVL C06051 V=8.0
MOVL C06052 V=8.0
MOVL C06053 V=8.0
MOVL C06054 V=8.0
MOVL C06055 V=8.0
MOVL C06056 V=8.0
MOVL C06057 V=8.0
MOVL C06058 V=8.0
MOVL C06059 V=8.0
MOVL C06060 V=8.0
MOVL C06061 V=8.0
MOVL C06062 V=8.0
MOVL C06063 V=8.0
MOVL C06064 V=8.0
MOVL C06065 V=8.0
MOVL C06066 V=8.0
MOVL C06067 V=8.0
MOVL C06068 V=8.0
MOVL C06069 V=8.0
MOVL C06070 V=8.0
MOVL C06071 V=8.0
MOVL C06072 V=8.0
MOVL C06073 V=8.0
MOVL C06074 V=8.0
MOVL C06075 V=8.0
MOVL C06076 V=8.0
MOVL C06077 V=8.0
MOVL C06078 V=8.0
MOVL C06079 V=8.0
MOVL C06080 V=8.0
MOVL C06081 V=8.0
MOVL C06082 V=8.0
MOVL C06083 V=8.0
MOVL C06084 V=8.0
MOVL C06085 V=8.0
MOVL C06086 V=8.0
MOVL C06087 V=8.0
MOVL C06088 V=8.0
MOVL C06089 V=8.0
MOVL C06090 V=8.0
MOVL C06091 V=8.0
MOVL C06092 V=8.0
MOVL C06093 V=8.0
MOVL C06094 V=8.0
MOVL C06095 V=8.0
MOVL C06096 V=8.0
MOVL C06097 V=8.0
MOVL C06098 V=8.0
MOVL C06099 V=8.0
MOVL C06100 V=8.0
MOVL C06101 V=8.0
MOVL C06102 V=8.0
MOVJ C06103 VJ=0.78
MOVL C06104 V=8.0
MOVL C06105 V=8.0
MOVL C06106 V=8.0
MOVL C06107 V=8.0
MOVL C06108 V=8.0
MOVL C06109 V=8.0
MOVL C06110 V=8.0
MOVL C06111 V=8.0
MOVL C06112 V=8.0
MOVL C06113 V=8.0
MOVL C06114 V=8.0
MOVL C06115 V=8.0
MOVL C06116 V=8.0
MOVL C06117 V=8.0
MOVL C06118 V=8.0
MOVL C06119 V=8.0
MOVL C06120 V=8.0
MOVL C06121 V=8.0
MOVL C06122 V=8.0
MOVL C06123 V=8.0
MOVL C06124 V=8.0
MOVJ C06125 VJ=0.78
MOVJ C06126 VJ=0.78
MOVL C06127 V=11.7
TIMER T=2.00
MOVL C06128 V=11.7
MOVJ C06129 VJ=0.78
MOVJ C06130 VJ=0.78
MOVL C06131 V=8.0
MOVL C06132 V=8.0
MOVL C06133 V=8.0
MOVL C06134 V=8.0
MOVL C06135 V=8.0
MOVL C06136 V=8.0
MOVL C06137 V=8.0
MOVL C06138 V=8.0
MOVL C06139 V=8.0
MOVL C06140 V=8.0
MOVL C06141 V=8.0
MOVL C06142 V=8.0
MOVL C06143 V=8.0
MOVL C06144 V=8.0
MOVL C06145 V=8.0
MOVL C06146 V=8.0
MOVL C06147 V=8.0
MOVL C06148 V=8.0
MOVL C06149 V=8.0
MOVL C06150 V=8.0
MOVL C06151 V=8.0
MOVL C06152 V=8.0
MOVL C06153 V=8.0
MOVL C06154 V=8.0
MOVL C06155 V=8.0
MOVL C06156 V=8.0
MOVL C06157 V=8.0
MOVL C06158 V=8.0
MOVL C06159 V=8.0
MOVL C06160 V=8.0
MOVL C06161 V=8.0
MOVL C06162 V=8.0
MOVL C06163 V=8.0
MOVL C06164 V=8.0
MOVL C06165 V=8.0
MOVL C06166 V=8.0
MOVL C06167 V=8.0
MOVL C06168 V=8.0
MOVL C06169 V=8.0
MOVL C06170 V=8.0
MOVL C06171 V=8.0
MOVL C06172 V=8.0
MOVJ C06173 VJ=0.78
MOVL C06174 V=8.0
MOVL C06175 V=8.0
MOVL C06176 V=8.0
MOVL C06177 V=8.0
MOVL C06178 V=8.0
MOVL C06179 V=8.0
MOVL C06180 V=8.0
MOVL C06181 V=8.0
MOVL C06182 V=8.0
MOVL C06183 V=8.0
MOVL C06184 V=8.0
MOVL C06185 V=8.0
MOVL C06186 V=8.0
MOVL C06187 V=8.0
MOVL C06188 V=8.0
MOVL C06189 V=8.0
MOVL C06190 V=8.0
MOVL C06191 V=8.0
MOVL C06192 V=8.0
MOVL C06193 V=8.0
MOVL C06194 V=8.0
MOVL C06195 V=8.0
MOVL C06196 V=8.0
MOVL C06197 V=8.0
MOVL C06198 V=8.0
MOVL C06199 V=8.0
MOVL C06200 V=8.0
MOVL C06201 V=8.0
MOVL C06202 V=8.0
MOVL C06203 V=8.0
MOVL C06204 V=8.0
MOVL C06205 V=8.0
MOVL C06206 V=8.0
MOVL C06207 V=8.0
MOVL C06208 V=8.0
MOVL C06209 V=8.0
MOVL C06210 V=8.0
MOVL C06211 V=8.0
MOVL C06212 V=8.0
MOVL C06213 V=8.0
MOVL C06214 V=8.0
MOVL C06215 V=8.0
MOVL C06216 V=8.0
MOVL C06217 V=8.0
MOVL C06218 V=8.0
MOVL C06219 V=8.0
MOVL C06220 V=8.0
MOVL C06221 V=8.0
MOVL C06222 V=8.0
MOVL C06223 V=8.0
MOVL C06224 V=8.0
MOVL C06225 V=8.0
MOVL C06226 V=8.0
MOVL C06227 V=8.0
MOVL C06228 V=8.0
MOVL C06229 V=8.0
MOVL C06230 V=8.0
MOVL C06231 V=8.0
MOVL C06232 V=8.0
MOVL C06233 V=8.0
MOVL C06234 V=8.0
MOVL C06235 V=8.0
MOVJ C06236 VJ=0.78
MOVL C06237 V=8.0
MOVL C06238 V=8.0
MOVL C06239 V=8.0
MOVL C06240 V=8.0
MOVL C06241 V=8.0
MOVL C06242 V=8.0
MOVL C06243 V=8.0
MOVL C06244 V=8.0
MOVL C06245 V=8.0
MOVL C06246 V=8.0
MOVL C06247 V=8.0
MOVL C06248 V=8.0
MOVL C06249 V=8.0
MOVL C06250 V=8.0
MOVL C06251 V=8.0
MOVL C06252 V=8.0
MOVL C06253 V=8.0
MOVL C06254 V=8.0
MOVL C06255 V=8.0
MOVL C06256 V=8.0
MOVL C06257 V=8.0
MOVL C06258 V=8.0
MOVL C06259 V=8.0
MOVL C06260 V=8.0
MOVL C06261 V=8.0
MOVL C06262 V=8.0
MOVL C06263 V=8.0
MOVL C06264 V=8.0
MOVL C06265 V=8.0
MOVL C06266 V=8.0
MOVL C06267 V=8.0
MOVL C06268 V=8.0
MOVL C06269 V=8.0
MOVL C06270 V=8.0
MOVL C06271 V=8.0
MOVL C06272 V=8.0
MOVL C06273 V=8.0
MOVL C06274 V=8.0
MOVL C06275 V=8.0
MOVL C06276 V=8.0
MOVL C06277 V=8.0
MOVL C06278 V=8.0
MOVL C06279 V=8.0
MOVL C06280 V=8.0
MOVL C06281 V=8.0
MOVL C06282 V=8.0
MOVL C06283 V=8.0
MOVL C06284 V=8.0
MOVL C06285 V=8.0
MOVL C06286 V=8.0
MOVL C06287 V=8.0
MOVL C06288 V=8.0
MOVL C06289 V=8.0
MOVL C06290 V=8.0
MOVL C06291 V=8.0
MOVL C06292 V=8.0
MOVL C06293 V=8.0
MOVL C06294 V=8.0
MOVL C06295 V=8.0
MOVL C06296 V=8.0
MOVL C06297 V=8.0
MOVJ C06298 VJ=0.78
MOVJ C06299 VJ=0.78
MOVL C06300 V=11.7
TIMER T=2.00
MOVL C06301 V=11.7
MOVJ C06302 VJ=0.78
MOVJ C06303 VJ=0.78
MOVL C06304 V=8.0
MOVL C06305 V=8.0
MOVJ C06306 VJ=0.78
MOVL C06307 V=8.0
MOVL C06308 V=8.0
MOVL C06309 V=8.0
MOVL C06310 V=8.0
MOVL C06311 V=8.0
MOVL C06312 V=8.0
MOVL C06313 V=8.0
MOVL C06314 V=8.0
MOVL C06315 V=8.0
MOVL C06316 V=8.0
MOVL C06317 V=8.0
MOVL C06318 V=8.0
MOVL C06319 V=8.0
MOVL C06320 V=8.0
MOVL C06321 V=8.0
MOVL C06322 V=8.0
MOVL C06323 V=8.0
MOVL C06324 V=8.0
MOVL C06325 V=8.0
MOVL C06326 V=8.0
MOVL C06327 V=8.0
MOVL C06328 V=8.0
MOVL C06329 V=8.0
MOVL C06330 V=8.0
MOVL C06331 V=8.0
MOVL C06332 V=8.0
MOVL C06333 V=8.0
MOVL C06334 V=8.0
MOVL C06335 V=8.0
MOVL C06336 V=8.0
MOVL C06337 V=8.0
MOVL C06338 V=8.0
MOVL C06339 V=8.0
MOVL C06340 V=8.0
MOVL C06341 V=8.0
MOVL C06342 V=8.0
MOVL C06343 V=8.0
MOVL C06344 V=8.0
MOVL C06345 V=8.0
MOVL C06346 V=8.0
MOVL C06347 V=8.0
MOVL C06348 V=8.0
MOVL C06349 V=8.0
MOVL C06350 V=8.0
MOVL C06351 V=8.0
MOVL C06352 V=8.0
MOVL C06353 V=8.0
MOVL C06354 V=8.0
MOVL C06355 V=8.0
MOVL C06356 V=8.0
MOVL C06357 V=8.0
MOVL C06358 V=8.0
MOVL C06359 V=8.0
MOVL C06360 V=8.0
MOVL C06361 V=8.0
MOVL C06362 V=8.0
MOVL C06363 V=8.0
MOVL C06364 V=8.0
MOVL C06365 V=8.0
MOVL C06366 V=8.0
MOVL C06367 V=8.0
MOVL C06368 V=8.0
MOVJ C06369 VJ=0.78
MOVL C06370 V=8.0
MOVL C06371 V=8.0
MOVL C06372 V=8.0
MOVL C06373 V=8.0
MOVL C06374 V=8.0
MOVL C06375 V=8.0
MOVL C06376 V=8.0
MOVL C06377 V=8.0
MOVL C06378 V=8.0
MOVL C06379 V=8.0
MOVL C06380 V=8.0
MOVL C06381 V=8.0
MOVL C06382 V=8.0
MOVL C06383 V=8.0
MOVL C06384 V=8.0
MOVL C06385 V=8.0
MOVL C06386 V=8.0
MOVL C06387 V=8.0
MOVL C06388 V=8.0
MOVL C06389 V=8.0
MOVL C06390 V=8.0
MOVL C06391 V=8.0
MOVL C06392 V=8.0
MOVL C06393 V=8.0
MOVL C06394 V=8.0
MOVL C06395 V=8.0
MOVL C06396 V=8.0
MOVL C06397 V=8.0
MOVL C06398 V=8.0
MOVL C06399 V=8.0
MOVL C06400 V=8.0
MOVL C06401 V=8.0
MOVL C06402 V=8.0
MOVL C06403 V=8.0
MOVL C06404 V=8.0
MOVL C06405 V=8.0
MOVL C06406 V=8.0
MOVL C06407 V=8.0
MOVL C06408 V=8.0
MOVL C06409 V=8.0
MOVL C06410 V=8.0
MOVL C06411 V=8.0
MOVL C06412 V=8.0
MOVL C06413 V=8.0
MOVL C06414 V=8.0
MOVL C06415 V=8.0
MOVL C06416 V=8.0
MOVL C06417 V=8.0
MOVL C06418 V=8.0
MOVL C06419 V=8.0
MOVL C06420 V=8.0
MOVL C06421 V=8.0
MOVL C06422 V=8.0
MOVL C06423 V=8.0
MOVL C06424 V=8.0
MOVL C06425 V=8.0
MOVL C06426 V=8.0
MOVL C06427 V=8.0
MOVL C06428 V=8.0
MOVL C06429 V=8.0
MOVL C06430 V=8.0
MOVL C06431 V=8.0
MOVJ C06432 VJ=0.78
MOVL C06433 V=8.0
MOVL C06434 V=8.0
MOVL C06435 V=8.0
MOVL C06436 V=8.0
MOVL C06437 V=8.0
MOVL C06438 V=8.0
MOVL C06439 V=8.0
MOVL C06440 V=8.0
MOVL C06441 V=8.0
MOVL C06442 V=8.0
MOVL C06443 V=8.0
MOVL C06444 V=8.0
MOVL C06445 V=8.0
MOVL C06446 V=8.0
MOVL C06447 V=8.0
MOVL C06448 V=8.0
MOVL C06449 V=8.0
MOVL C06450 V=8.0
MOVL C06451 V=8.0
MOVL C06452 V=8.0
MOVL C06453 V=8.0
MOVL C06454 V=8.0
MOVL C06455 V=8.0
MOVL C06456 V=8.0
MOVL C06457 V=8.0
MOVL C06458 V=8.0
MOVL C06459 V=8.0
MOVL C06460 V=8.0
MOVL C06461 V=8.0
MOVL C06462 V=8.0
MOVL C06463 V=8.0
MOVL C06464 V=8.0
MOVL C06465 V=8.0
MOVL C06466 V=8.0
MOVL C06467 V=8.0
MOVL C06468 V=8.0
MOVL C06469 V=8.0
MOVL C06470 V=8.0
MOVL C06471 V=8.0
MOVL C06472 V=8.0
MOVL C06473 V=8.0
MOVJ C06474 VJ=0.78
MOVJ C06475 VJ=0.78
MOVL C06476 V=11.7
TIMER T=2.00
MOVL C06477 V=11.7
MOVJ C06478 VJ=0.78
MOVJ C06479 VJ=0.78
MOVL C06480 V=8.0
MOVL C06481 V=8.0
MOVL C06482 V=8.0
MOVL C06483 V=8.0
MOVL C06484 V=8.0
MOVL C06485 V=8.0
MOVL C06486 V=8.0
MOVL C06487 V=8.0
MOVL C06488 V=8.0
MOVL C06489 V=8.0
MOVL C06490 V=8.0
MOVL C06491 V=8.0
MOVL C06492 V=8.0
MOVL C06493 V=8.0
MOVL C06494 V=8.0
MOVL C06495 V=8.0
MOVL C06496 V=8.0
MOVL C06497 V=8.0
MOVL C06498 V=8.0
MOVL C06499 V=8.0
MOVL C06500 V=8.0
MOVL C06501 V=8.0
MOVJ C06502 VJ=0.78
MOVL C06503 V=8.0
MOVL C06504 V=8.0
MOVL C06505 V=8.0
MOVL C06506 V=8.0
MOVL C06507 V=8.0
MOVL C06508 V=8.0
MOVL C06509 V=8.0
MOVL C06510 V=8.0
MOVL C06511 V=8.0
MOVL C06512 V=8.0
MOVL C06513 V=8.0
MOVL C06514 V=8.0
MOVL C06515 V=8.0
MOVL C06516 V=8.0
MOVL C06517 V=8.0
MOVL C06518 V=8.0
MOVL C06519 V=8.0
MOVL C06520 V=8.0
MOVL C06521 V=8.0
MOVL C06522 V=8.0
MOVL C06523 V=8.0
MOVL C06524 V=8.0
MOVL C06525 V=8.0
MOVL C06526 V=8.0
MOVL C06527 V=8.0
MOVL C06528 V=8.0
MOVL C06529 V=8.0
MOVL C06530 V=8.0
MOVL C06531 V=8.0
MOVL C06532 V=8.0
MOVL C06533 V=8.0
MOVL C06534 V=8.0
MOVL C06535 V=8.0
MOVL C06536 V=8.0
MOVL C06537 V=8.0
MOVL C06538 V=8.0
MOVL C06539 V=8.0
MOVL C06540 V=8.0
MOVL C06541 V=8.0
MOVL C06542 V=8.0
MOVL C06543 V=8.0
MOVL C06544 V=8.0
MOVL C06545 V=8.0
MOVL C06546 V=8.0
MOVL C06547 V=8.0
MOVL C06548 V=8.0
MOVL C06549 V=8.0
MOVL C06550 V=8.0
MOVL C06551 V=8.0
MOVL C06552 V=8.0
MOVL C06553 V=8.0
MOVL C06554 V=8.0
MOVL C06555 V=8.0
MOVL C06556 V=8.0
MOVL C06557 V=8.0
MOVL C06558 V=8.0
MOVL C06559 V=8.0
MOVL C06560 V=8.0
MOVL C06561 V=8.0
MOVL C06562 V=8.0
MOVL C06563 V=8.0
MOVL C06564 V=8.0
MOVJ C06565 VJ=0.78
MOVL C06566 V=8.0
MOVL C06567 V=8.0
MOVL C06568 V=8.0
MOVL C06569 V=8.0
MOVL C06570 V=8.0
MOVL C06571 V=8.0
MOVL C06572 V=8.0
MOVL C06573 V=8.0
MOVL C06574 V=8.0
MOVL C06575 V=8.0
MOVL C06576 V=8.0
MOVL C06577 V=8.0
MOVL C06578 V=8.0
MOVL C06579 V=8.0
MOVL C06580 V=8.0
MOVL C06581 V=8.0
MOVL C06582 V=8.0
MOVL C06583 V=8.0
MOVL C06584 V=8.0
MOVL C06585 V=8.0
MOVL C06586 V=8.0
MOVL C06587 V=8.0
MOVL C06588 V=8.0
MOVL C06589 V=8.0
MOVL C06590 V=8.0
MOVL C06591 V=8.0
MOVL C06592 V=8.0
MOVL C06593 V=8.0
MOVL C06594 V=8.0
MOVL C06595 V=8.0
MOVL C06596 V=8.0
MOVL C06597 V=8.0
MOVL C06598 V=8.0
MOVL C06599 V=8.0
MOVL C06600 V=8.0
MOVL C06601 V=8.0
MOVL C06602 V=8.0
MOVL C06603 V=8.0
MOVL C06604 V=8.0
MOVL C06605 V=8.0
MOVL C06606 V=8.0
MOVL C06607 V=8.0
MOVL C06608 V=8.0
MOVL C06609 V=8.0
MOVL C06610 V=8.0
MOVL C06611 V=8.0
MOVL C06612 V=8.0
MOVL C06613 V=8.0
MOVL C06614 V=8.0
MOVL C06615 V=8.0
MOVL C06616 V=8.0
MOVL C06617 V=8.0
MOVL C06618 V=8.0
MOVL C06619 V=8.0
MOVL C06620 V=8.0
MOVL C06621 V=8.0
MOVL C06622 V=8.0
MOVL C06623 V=8.0
MOVL C06624 V=8.0
MOVL C06625 V=8.0
MOVL C06626 V=8.0
MOVL C06627 V=8.0
MOVJ C06628 VJ=0.78
MOVL C06629 V=8.0
MOVL C06630 V=8.0
MOVL C06631 V=8.0
MOVL C06632 V=8.0
MOVL C06633 V=8.0
MOVL C06634 V=8.0
MOVL C06635 V=8.0
MOVL C06636 V=8.0
MOVL C06637 V=8.0
MOVL C06638 V=8.0
MOVL C06639 V=8.0
MOVL C06640 V=8.0
MOVL C06641 V=8.0
MOVL C06642 V=8.0
MOVL C06643 V=8.0
MOVL C06644 V=8.0
MOVL C06645 V=8.0
MOVL C06646 V=8.0
MOVL C06647 V=8.0
MOVL C06648 V=8.0
MOVL C06649 V=8.0
MOVJ C06650 VJ=0.78
MOVJ C06651 VJ=0.78
MOVL C06652 V=11.7
TIMER T=2.00
MOVL C06653 V=11.7
MOVJ C06654 VJ=0.78
MOVJ C06655 VJ=0.78
MOVL C06656 V=8.0
MOVL C06657 V=8.0
MOVL C06658 V=8.0
MOVL C06659 V=8.0
MOVL C06660 V=8.0
MOVL C06661 V=8.0
MOVL C06662 V=8.0
MOVL C06663 V=8.0
MOVL C06664 V=8.0
MOVL C06665 V=8.0
MOVL C06666 V=8.0
MOVL C06667 V=8.0
MOVL C06668 V=8.0
MOVL C06669 V=8.0
MOVL C06670 V=8.0
MOVL C06671 V=8.0
MOVL C06672 V=8.0
MOVL C06673 V=8.0
MOVL C06674 V=8.0
MOVL C06675 V=8.0
MOVL C06676 V=8.0
MOVL C06677 V=8.0
MOVL C06678 V=8.0
MOVL C06679 V=8.0
MOVL C06680 V=8.0
MOVL C06681 V=8.0
MOVL C06682 V=8.0
MOVL C06683 V=8.0
MOVL C06684 V=8.0
MOVL C06685 V=8.0
MOVL C06686 V=8.0
MOVL C06687 V=8.0
MOVL C06688 V=8.0
MOVL C06689 V=8.0
MOVL C06690 V=8.0
MOVL C06691 V=8.0
MOVL C06692 V=8.0
MOVL C06693 V=8.0
MOVL C06694 V=8.0
MOVL C06695 V=8.0
MOVL C06696 V=8.0
MOVL C06697 V=8.0
MOVJ C06698 VJ=0.78
MOVL C06699 V=8.0
MOVL C06700 V=8.0
MOVL C06701 V=8.0
MOVL C06702 V=8.0
MOVL C06703 V=8.0
MOVL C06704 V=8.0
MOVL C06705 V=8.0
MOVL C06706 V=8.0
MOVL C06707 V=8.0
MOVL C06708 V=8.0
MOVL C06709 V=8.0
MOVL C06710 V=8.0
MOVL C06711 V=8.0
MOVL C06712 V=8.0
MOVL C06713 V=8.0
MOVL C06714 V=8.0
MOVL C06715 V=8.0
MOVL C06716 V=8.0
MOVL C06717 V=8.0
MOVL C06718 V=8.0
MOVL C06719 V=8.0
MOVL C06720 V=8.0
MOVL C06721 V=8.0
MOVL C06722 V=8.0
MOVL C06723 V=8.0
MOVL C06724 V=8.0
MOVL C06725 V=8.0
MOVL C06726 V=8.0
MOVL C06727 V=8.0
MOVL C06728 V=8.0
MOVL C06729 V=8.0
MOVL C06730 V=8.0
MOVL C06731 V=8.0
MOVL C06732 V=8.0
MOVL C06733 V=8.0
MOVL C06734 V=8.0
MOVL C06735 V=8.0
MOVL C06736 V=8.0
MOVL C06737 V=8.0
MOVL C06738 V=8.0
MOVL C06739 V=8.0
MOVL C06740 V=8.0
MOVL C06741 V=8.0
MOVL C06742 V=8.0
MOVL C06743 V=8.0
MOVL C06744 V=8.0
MOVL C06745 V=8.0
MOVL C06746 V=8.0
MOVL C06747 V=8.0
MOVL C06748 V=8.0
MOVL C06749 V=8.0
MOVL C06750 V=8.0
MOVL C06751 V=8.0
MOVL C06752 V=8.0
MOVL C06753 V=8.0
MOVL C06754 V=8.0
MOVL C06755 V=8.0
MOVL C06756 V=8.0
MOVL C06757 V=8.0
MOVL C06758 V=8.0
MOVL C06759 V=8.0
MOVL C06760 V=8.0
MOVJ C06761 VJ=0.78
MOVL C06762 V=8.0
MOVL C06763 V=8.0
MOVL C06764 V=8.0
MOVL C06765 V=8.0
MOVL C06766 V=8.0
MOVL C06767 V=8.0
MOVL C06768 V=8.0
MOVL C06769 V=8.0
MOVL C06770 V=8.0
MOVL C06771 V=8.0
MOVL C06772 V=8.0
MOVL C06773 V=8.0
MOVL C06774 V=8.0
MOVL C06775 V=8.0
MOVL C06776 V=8.0
MOVL C06777 V=8.0
MOVL C06778 V=8.0
MOVL C06779 V=8.0
MOVL C06780 V=8.0
MOVL C06781 V=8.0
MOVL C06782 V=8.0
MOVL C06783 V=8.0
MOVL C06784 V=8.0
MOVL C06785 V=8.0
MOVL C06786 V=8.0
MOVL C06787 V=8.0
MOVL C06788 V=8.0
MOVL C06789 V=8.0
MOVL C06790 V=8.0
MOVL C06791 V=8.0
MOVL C06792 V=8.0
MOVL C06793 V=8.0
MOVL C06794 V=8.0
MOVL C06795 V=8.0
MOVL C06796 V=8.0
MOVL C06797 V=8.0
MOVL C06798 V=8.0
MOVL C06799 V=8.0
MOVL C06800 V=8.0
MOVL C06801 V=8.0
MOVL C06802 V=8.0
MOVL C06803 V=8.0
MOVL C06804 V=8.0
MOVL C06805 V=8.0
MOVL C06806 V=8.0
MOVL C06807 V=8.0
MOVL C06808 V=8.0
MOVL C06809 V=8.0
MOVL C06810 V=8.0
MOVL C06811 V=8.0
MOVL C06812 V=8.0
MOVL C06813 V=8.0
MOVL C06814 V=8.0
MOVL C06815 V=8.0
MOVL C06816 V=8.0
MOVL C06817 V=8.0
MOVL C06818 V=8.0
MOVL C06819 V=8.0
MOVL C06820 V=8.0
MOVL C06821 V=8.0
MOVL C06822 V=8.0
MOVJ C06823 VJ=0.78
MOVJ C06824 VJ=0.78
MOVL C06825 V=11.7
TIMER T=2.00
MOVL C06826 V=11.7
MOVJ C06827 VJ=0.78
MOVJ C06828 VJ=0.78
MOVL C06829 V=8.0
MOVL C06830 V=8.0
MOVJ C06831 VJ=0.78
MOVL C06832 V=8.0
MOVL C06833 V=8.0
MOVL C06834 V=8.0
MOVL C06835 V=8.0
MOVL C06836 V=8.0
MOVL C06837 V=8.0
MOVL C06838 V=8.0
MOVL C06839 V=8.0
MOVL C06840 V=8.0
MOVL C06841 V=8.0
MOVL C06842 V=8.0
MOVL C06843 V=8.0
MOVL C06844 V=8.0
MOVL C06845 V=8.0
MOVL C06846 V=8.0
MOVL C06847 V=8.0
MOVL C06848 V=8.0
MOVL C06849 V=8.0
MOVL C06850 V=8.0
MOVL C06851 V=8.0
MOVL C06852 V=8.0
MOVL C06853 V=8.0
MOVL C06854 V=8.0
MOVL C06855 V=8.0
MOVL C06856 V=8.0
MOVL C06857 V=8.0
MOVL C06858 V=8.0
MOVL C06859 V=8.0
MOVL C06860 V=8.0
MOVL C06861 V=8.0
MOVL C06862 V=8.0
MOVL C06863 V=8.0
MOVL C06864 V=8.0
MOVL C06865 V=8.0
MOVL C06866 V=8.0
MOVL C06867 V=8.0
MOVL C06868 V=8.0
MOVL C06869 V=8.0
MOVL C06870 V=8.0
MOVL C06871 V=8.0
MOVL C06872 V=8.0
MOVL C06873 V=8.0
MOVL C06874 V=8.0
MOVL C06875 V=8.0
MOVL C06876 V=8.0
MOVL C06877 V=8.0
MOVL C06878 V=8.0
MOVL C06879 V=8.0
MOVL C06880 V=8.0
MOVL C06881 V=8.0
MOVL C06882 V=8.0
MOVL C06883 V=8.0
MOVL C06884 V=8.0
MOVL C06885 V=8.0
MOVL C06886 V=8.0
MOVL C06887 V=8.0
MOVL C06888 V=8.0
MOVL C06889 V=8.0
MOVL C06890 V=8.0
MOVL C06891 V=8.0
MOVL C06892 V=8.0
MOVL C06893 V=8.0
MOVJ C06894 VJ=0.78
MOVL C06895 V=8.0
MOVL C06896 V=8.0
MOVL C06897 V=8.0
MOVL C06898 V=8.0
MOVL C06899 V=8.0
MOVL C06900 V=8.0
MOVL C06901 V=8.0
MOVL C06902 V=8.0
MOVL C06903 V=8.0
MOVL C06904 V=8.0
MOVL C06905 V=8.0
MOVL C06906 V=8.0
MOVL C06907 V=8.0
MOVL C06908 V=8.0
MOVL C06909 V=8.0
MOVL C06910 V=8.0
MOVL C06911 V=8.0
MOVL C06912 V=8.0
MOVL C06913 V=8.0
MOVL C06914 V=8.0
MOVL C06915 V=8.0
MOVL C06916 V=8.0
MOVL C06917 V=8.0
MOVL C06918 V=8.0
MOVL C06919 V=8.0
MOVL C06920 V=8.0
MOVL C06921 V=8.0
MOVL C06922 V=8.0
MOVL C06923 V=8.0
MOVL C06924 V=8.0
MOVL C06925 V=8.0
MOVL C06926 V=8.0
MOVL C06927 V=8.0
MOVL C06928 V=8.0
MOVL C06929 V=8.0
MOVL C06930 V=8.0
MOVL C06931 V=8.0
MOVL C06932 V=8.0
MOVL C06933 V=8.0
MOVL C06934 V=8.0
MOVL C06935 V=8.0
MOVL C06936 V=8.0
MOVL C06937 V=8.0
MOVL C06938 V=8.0
MOVL C06939 V=8.0
MOVL C06940 V=8.0
MOVL C06941 V=8.0
MOVL C06942 V=8.0
MOVL C06943 V=8.0
MOVL C06944 V=8.0
MOVL C06945 V=8.0
MOVL C06946 V=8.0
MOVL C06947 V=8.0
MOVL C06948 V=8.0
MOVL C06949 V=8.0
MOVL C06950 V=8.0
MOVL C06951 V=8.0
MOVL C06952 V=8.0
MOVL C06953 V=8.0
MOVL C06954 V=8.0
MOVL C06955 V=8.0
MOVL C06956 V=8.0
MOVJ C06957 VJ=0.78
MOVL C06958 V=8.0
MOVL C06959 V=8.0
MOVL C06960 V=8.0
MOVL C06961 V=8.0
MOVL C06962 V=8.0
MOVL C06963 V=8.0
MOVL C06964 V=8.0
MOVL C06965 V=8.0
MOVL C06966 V=8.0
MOVL C06967 V=8.0
MOVL C06968 V=8.0
MOVL C06969 V=8.0
MOVL C06970 V=8.0
MOVL C06971 V=8.0
MOVL C06972 V=8.0
MOVL C06973 V=8.0
MOVL C06974 V=8.0
MOVL C06975 V=8.0
MOVL C06976 V=8.0
MOVL C06977 V=8.0
MOVL C06978 V=8.0
MOVL C06979 V=8.0
MOVL C06980 V=8.0
MOVL C06981 V=8.0
MOVL C06982 V=8.0
MOVL C06983 V=8.0
MOVL C06984 V=8.0
MOVL C06985 V=8.0
MOVL C06986 V=8.0
MOVL C06987 V=8.0
MOVL C06988 V=8.0
MOVL C06989 V=8.0
MOVL C06990 V=8.0
MOVL C06991 V=8.0
MOVL C06992 V=8.0
MOVL C06993 V=8.0
MOVL C06994 V=8.0
MOVL C06995 V=8.0
MOVL C06996 V=8.0
MOVL C06997 V=8.0
MOVL C06998 V=8.0
MOVJ C06999 VJ=0.78
MOVJ C07000 VJ=0.78
MOVL C07001 V=11.7
TIMER T=2.00
MOVL C07002 V=11.7
MOVJ C07003 VJ=0.78
MOVJ C07004 VJ=0.78
MOVL C07005 V=8.0
MOVL C07006 V=8.0
MOVL C07007 V=8.0
MOVL C07008 V=8.0
MOVL C07009 V=8.0
MOVL C07010 V=8.0
MOVL C07011 V=8.0
MOVL C07012 V=8.0
MOVL C07013 V=8.0
MOVL C07014 V=8.0
MOVL C07015 V=8.0
MOVL C07016 V=8.0
MOVL C07017 V=8.0
MOVL C07018 V=8.0
MOVL C07019 V=8.0
MOVL C07020 V=8.0
MOVL C07021 V=8.0
MOVL C07022 V=8.0
MOVL C07023 V=8.0
MOVL C07024 V=8.0
MOVL C07025 V=8.0
MOVL C07026 V=8.0
MOVJ C07027 VJ=0.78
MOVL C07028 V=8.0
MOVL C07029 V=8.0
MOVL C07030 V=8.0
MOVL C07031 V=8.0
MOVL C07032 V=8.0
MOVL C07033 V=8.0
MOVL C07034 V=8.0
MOVL C07035 V=8.0
MOVL C07036 V=8.0
MOVL C07037 V=8.0
MOVL C07038 V=8.0
MOVL C07039 V=8.0
MOVL C07040 V=8.0
MOVL C07041 V=8.0
MOVL C07042 V=8.0
MOVL C07043 V=8.0
MOVL C07044 V=8.0
MOVL C07045 V=8.0
MOVL C07046 V=8.0
MOVL C07047 V=8.0
MOVL C07048 V=8.0
MOVL C07049 V=8.0
MOVL C07050 V=8.0
MOVL C07051 V=8.0
MOVL C07052 V=8.0
MOVL C07053 V=8.0
MOVL C07054 V=8.0
MOVL C07055 V=8.0
MOVL C07056 V=8.0
MOVL C07057 V=8.0
MOVL C07058 V=8.0
MOVL C07059 V=8.0
MOVL C07060 V=8.0
MOVL C07061 V=8.0
MOVL C07062 V=8.0
MOVL C07063 V=8.0
MOVL C07064 V=8.0
MOVL C07065 V=8.0
MOVL C07066 V=8.0
MOVL C07067 V=8.0
MOVL C07068 V=8.0
MOVL C07069 V=8.0
MOVL C07070 V=8.0
MOVL C07071 V=8.0
MOVL C07072 V=8.0
MOVL C07073 V=8.0
MOVL C07074 V=8.0
MOVL C07075 V=8.0
MOVL C07076 V=8.0
MOVL C07077 V=8.0
MOVL C07078 V=8.0
MOVL C07079 V=8.0
MOVL C07080 V=8.0
MOVL C07081 V=8.0
MOVL C07082 V=8.0
MOVL C07083 V=8.0
MOVL C07084 V=8.0
MOVL C07085 V=8.0
MOVL C07086 V=8.0
MOVL C07087 V=8.0
MOVL C07088 V=8.0
MOVL C07089 V=8.0
MOVJ C07090 VJ=0.78
MOVL C07091 V=8.0
MOVL C07092 V=8.0
MOVL C07093 V=8.0
MOVL C07094 V=8.0
MOVL C07095 V=8.0
MOVL C07096 V=8.0
MOVL C07097 V=8.0
MOVL C07098 V=8.0
MOVL C07099 V=8.0
MOVL C07100 V=8.0
MOVL C07101 V=8.0
MOVL C07102 V=8.0
MOVL C07103 V=8.0
MOVL C07104 V=8.0
MOVL C07105 V=8.0
MOVL C07106 V=8.0
MOVL C07107 V=8.0
MOVL C07108 V=8.0
MOVL C07109 V=8.0
MOVL C07110 V=8.0
MOVL C07111 V=8.0
MOVL C07112 V=8.0
MOVL C07113 V=8.0
MOVL C07114 V=8.0
MOVL C07115 V=8.0
MOVL C07116 V=8.0
MOVL C07117 V=8.0
MOVL C07118 V=8.0
MOVL C07119 V=8.0
MOVL C07120 V=8.0
MOVL C07121 V=8.0
MOVL C07122 V=8.0
MOVL C07123 V=8.0
MOVL C07124 V=8.0
MOVL C07125 V=8.0
MOVL C07126 V=8.0
MOVL C07127 V=8.0
MOVL C07128 V=8.0
MOVL C07129 V=8.0
MOVL C07130 V=8.0
MOVL C07131 V=8.0
MOVL C07132 V=8.0
MOVL C07133 V=8.0
MOVL C07134 V=8.0
MOVL C07135 V=8.0
MOVL C07136 V=8.0
MOVL C07137 V=8.0
MOVL C07138 V=8.0
MOVL C07139 V=8.0
MOVL C07140 V=8.0
MOVL C07141 V=8.0
MOVL C07142 V=8.0
MOVL C07143 V=8.0
MOVL C07144 V=8.0
MOVL C07145 V=8.0
MOVL C07146 V=8.0
MOVL C07147 V=8.0
MOVL C07148 V=8.0
MOVL C07149 V=8.0
MOVL C07150 V=8.0
MOVL C07151 V=8.0
MOVL C07152 V=8.0
MOVJ C07153 VJ=0.78
MOVL C07154 V=8.0
MOVL C07155 V=8.0
MOVL C07156 V=8.0
MOVL C07157 V=8.0
MOVL C07158 V=8.0
MOVL C07159 V=8.0
MOVL C07160 V=8.0
MOVL C07161 V=8.0
MOVL C07162 V=8.0
MOVL C07163 V=8.0
MOVL C07164 V=8.0
MOVL C07165 V=8.0
MOVL C07166 V=8.0
MOVL C07167 V=8.0
MOVL C07168 V=8.0
MOVL C07169 V=8.0
MOVL C07170 V=8.0
MOVL C07171 V=8.0
MOVL C07172 V=8.0
MOVL C07173 V=8.0
MOVL C07174 V=8.0
MOVJ C07175 VJ=0.78
MOVJ C07176 VJ=0.78
MOVL C07177 V=11.7
TIMER T=2.00
MOVL C07178 V=11.7
MOVJ C07179 VJ=0.78
MOVJ C07180 VJ=0.78
MOVL C07181 V=8.0
MOVL C07182 V=8.0
MOVL C07183 V=8.0
MOVL C07184 V=8.0
MOVL C07185 V=8.0
MOVL C07186 V=8.0
MOVL C07187 V=8.0
MOVL C07188 V=8.0
MOVL C07189 V=8.0
MOVL C07190 V=8.0
MOVL C07191 V=8.0
MOVL C07192 V=8.0
MOVL C07193 V=8.0
MOVL C07194 V=8.0
MOVL C07195 V=8.0
MOVL C07196 V=8.0
MOVL C07197 V=8.0
MOVL C07198 V=8.0
MOVL C07199 V=8.0
MOVL C07200 V=8.0
MOVL C07201 V=8.0
MOVL C07202 V=8.0
MOVL C07203 V=8.0
MOVL C07204 V=8.0
MOVL C07205 V=8.0
MOVL C07206 V=8.0
MOVL C07207 V=8.0
MOVL C07208 V=8.0
MOVL C07209 V=8.0
MOVL C07210 V=8.0
MOVL C07211 V=8.0
MOVL C07212 V=8.0
MOVL C07213 V=8.0
MOVL C07214 V=8.0
MOVL C07215 V=8.0
MOVL C07216 V=8.0
MOVL C07217 V=8.0
MOVL C07218 V=8.0
MOVL C07219 V=8.0
MOVL C07220 V=8.0
MOVL C07221 V=8.0
MOVL C07222 V=8.0
MOVJ C07223 VJ=0.78
MOVL C07224 V=8.0
MOVL C07225 V=8.0
MOVL C07226 V=8.0
MOVL C07227 V=8.0
MOVL C07228 V=8.0
MOVL C07229 V=8.0
MOVL C07230 V=8.0
MOVL C07231 V=8.0
MOVL C07232 V=8.0
MOVL C07233 V=8.0
MOVL C07234 V=8.0
MOVL C07235 V=8.0
MOVL C07236 V=8.0
MOVL C07237 V=8.0
MOVL C07238 V=8.0
MOVL C07239 V=8.0
MOVL C07240 V=8.0
MOVL C07241 V=8.0
MOVL C07242 V=8.0
MOVL C07243 V=8.0
MOVL C07244 V=8.0
MOVL C07245 V=8.0
MOVL C07246 V=8.0
MOVL C07247 V=8.0
MOVL C07248 V=8.0
MOVL C07249 V=8.0
MOVL C07250 V=8.0
MOVL C07251 V=8.0
MOVL C07252 V=8.0
MOVL C07253 V=8.0
MOVL C07254 V=8.0
MOVL C07255 V=8.0
MOVL C07256 V=8.0
MOVL C07257 V=8.0
MOVL C07258 V=8.0
MOVL C07259 V=8.0
MOVL C07260 V=8.0
MOVL C07261 V=8.0
MOVL C07262 V=8.0
MOVL C07263 V=8.0
MOVL C07264 V=8.0
MOVL C07265 V=8.0
MOVL C07266 V=8.0
MOVL C07267 V=8.0
MOVL C07268 V=8.0
MOVL C07269 V=8.0
MOVL C07270 V=8.0
MOVL C07271 V=8.0
MOVL C07272 V=8.0
MOVL C07273 V=8.0
MOVL C07274 V=8.0
MOVL C07275 V=8.0
MOVL C07276 V=8.0
MOVL C07277 V=8.0
MOVL C07278 V=8.0
MOVL C07279 V=8.0
MOVL C07280 V=8.0
MOVL C07281 V=8.0
MOVL C07282 V=8.0
MOVL C07283 V=8.0
MOVL C07284 V=8.0
MOVL C07285 V=8.0
MOVJ C07286 VJ=0.78
MOVL C07287 V=8.0
MOVL C07288 V=8.0
MOVL C07289 V=8.0
MOVL C07290 V=8.0
MOVL C07291 V=8.0
MOVL C07292 V=8.0
MOVL C07293 V=8.0
MOVL C07294 V=8.0
MOVL C07295 V=8.0
MOVL C07296 V=8.0
MOVL C07297 V=8.0
MOVL C07298 V=8.0
MOVL C07299 V=8.0
MOVL C07300 V=8.0
MOVL C07301 V=8.0
MOVL C07302 V=8.0
MOVL C07303 V=8.0
MOVL C07304 V=8.0
MOVL C07305 V=8.0
MOVL C07306 V=8.0
MOVL C07307 V=8.0
MOVL C07308 V=8.0
MOVL C07309 V=8.0
MOVL C07310 V=8.0
MOVL C07311 V=8.0
MOVL C07312 V=8.0
MOVL C07313 V=8.0
MOVL C07314 V=8.0
MOVL C07315 V=8.0
MOVL C07316 V=8.0
MOVL C07317 V=8.0
MOVL C07318 V=8.0
MOVL C07319 V=8.0
MOVL C07320 V=8.0
MOVL C07321 V=8.0
MOVL C07322 V=8.0
MOVL C07323 V=8.0
MOVL C07324 V=8.0
MOVL C07325 V=8.0
MOVL C07326 V=8.0
MOVL C07327 V=8.0
MOVL C07328 V=8.0
MOVL C07329 V=8.0
MOVL C07330 V=8.0
MOVL C07331 V=8.0
MOVL C07332 V=8.0
MOVL C07333 V=8.0
MOVL C07334 V=8.0
MOVL C07335 V=8.0
MOVL C07336 V=8.0
MOVL C07337 V=8.0
MOVL C07338 V=8.0
MOVL C07339 V=8.0
MOVL C07340 V=8.0
MOVL C07341 V=8.0
MOVL C07342 V=8.0
MOVL C07343 V=8.0
MOVL C07344 V=8.0
MOVL C07345 V=8.0
MOVL C07346 V=8.0
MOVL C07347 V=8.0
MOVJ C07348 VJ=0.78
MOVJ C07349 VJ=0.78
MOVL C07350 V=11.7
TIMER T=2.00
MOVL C07351 V=11.7
MOVJ C07352 VJ=0.78
MOVJ C07353 VJ=0.78
MOVL C07354 V=8.0
MOVL C07355 V=8.0
MOVJ C07356 VJ=0.78
MOVL C07357 V=8.0
MOVL C07358 V=8.0
MOVL C07359 V=8.0
MOVL C07360 V=8.0
MOVL C07361 V=8.0
MOVL C07362 V=8.0
MOVL C07363 V=8.0
MOVL C07364 V=8.0
MOVL C07365 V=8.0
MOVL C07366 V=8.0
MOVL C07367 V=8.0
MOVL C07368 V=8.0
MOVL C07369 V=8.0
MOVL C07370 V=8.0
MOVL C07371 V=8.0
MOVL C07372 V=8.0
MOVL C07373 V=8.0
MOVL C07374 V=8.0
MOVL C07375 V=8.0
MOVL C07376 V=8.0
MOVL C07377 V=8.0
MOVL C07378 V=8.0
MOVL C07379 V=8.0
MOVL C07380 V=8.0
MOVL C07381 V=8.0
MOVL C07382 V=8.0
MOVL C07383 V=8.0
MOVL C07384 V=8.0
MOVL C07385 V=8.0
MOVL C07386 V=8.0
MOVL C07387 V=8.0
MOVL C07388 V=8.0
MOVL C07389 V=8.0
MOVL C07390 V=8.0
MOVL C07391 V=8.0
MOVL C07392 V=8.0
MOVL C07393 V=8.0
MOVL C07394 V=8.0
MOVL C07395 V=8.0
MOVL C07396 V=8.0
MOVL C07397 V=8.0
MOVL C07398 V=8.0
MOVL C07399 V=8.0
MOVL C07400 V=8.0
MOVL C07401 V=8.0
MOVL C07402 V=8.0
MOVL C07403 V=8.0
MOVL C07404 V=8.0
MOVL C07405 V=8.0
MOVL C07406 V=8.0
MOVL C07407 V=8.0
MOVL C07408 V=8.0
MOVL C07409 V=8.0
MOVL C07410 V=8.0
MOVL C07411 V=8.0
MOVL C07412 V=8.0
MOVL C07413 V=8.0
MOVL C07414 V=8.0
MOVL C07415 V=8.0
MOVL C07416 V=8.0
MOVL C07417 V=8.0
MOVL C07418 V=8.0
MOVJ C07419 VJ=0.78
MOVL C07420 V=8.0
MOVL C07421 V=8.0
MOVL C07422 V=8.0
MOVL C07423 V=8.0
MOVL C07424 V=8.0
MOVL C07425 V=8.0
MOVL C07426 V=8.0
MOVL C07427 V=8.0
MOVL C07428 V=8.0
MOVL C07429 V=8.0
MOVL C07430 V=8.0
MOVL C07431 V=8.0
MOVL C07432 V=8.0
MOVL C07433 V=8.0
MOVL C07434 V=8.0
MOVL C07435 V=8.0
MOVL C07436 V=8.0
MOVL C07437 V=8.0
MOVL C07438 V=8.0
MOVL C07439 V=8.0
MOVL C07440 V=8.0
MOVL C07441 V=8.0
MOVL C07442 V=8.0
MOVL C07443 V=8.0
MOVL C07444 V=8.0
MOVL C07445 V=8.0
MOVL C07446 V=8.0
MOVL C07447 V=8.0
MOVL C07448 V=8.0
MOVL C07449 V=8.0
MOVL C07450 V=8.0
MOVL C07451 V=8.0
MOVL C07452 V=8.0
MOVL C07453 V=8.0
MOVL C07454 V=8.0
MOVL C07455 V=8.0
MOVL C07456 V=8.0
MOVL C07457 V=8.0
MOVL C07458 V=8.0
MOVL C07459 V=8.0
MOVL C07460 V=8.0
MOVL C07461 V=8.0
MOVL C07462 V=8.0
MOVL C07463 V=8.0
MOVL C07464 V=8.0
MOVL C07465 V=8.0
MOVL C07466 V=8.0
MOVL C07467 V=8.0
MOVL C07468 V=8.0
MOVL C07469 V=8.0
MOVL C07470 V=8.0
MOVL C07471 V=8.0
MOVL C07472 V=8.0
MOVL C07473 V=8.0
MOVL C07474 V=8.0
MOVL C07475 V=8.0
MOVL C07476 V=8.0
MOVL C07477 V=8.0
MOVL C07478 V=8.0
MOVL C07479 V=8.0
MOVL C07480 V=8.0
MOVL C07481 V=8.0
MOVJ C07482 VJ=0.78
MOVL C07483 V=8.0
MOVL C07484 V=8.0
MOVL C07485 V=8.0
MOVL C07486 V=8.0
MOVL C07487 V=8.0
MOVL C07488 V=8.0
MOVL C07489 V=8.0
MOVL C07490 V=8.0
MOVL C07491 V=8.0
MOVL C07492 V=8.0
MOVL C07493 V=8.0
MOVL C07494 V=8.0
MOVL C07495 V=8.0
MOVL C07496 V=8.0
MOVL C07497 V=8.0
MOVL C07498 V=8.0
MOVL C07499 V=8.0
MOVL C07500 V=8.0
MOVL C07501 V=8.0
MOVL C07502 V=8.0
MOVL C07503 V=8.0
MOVL C07504 V=8.0
MOVL C07505 V=8.0
MOVL C07506 V=8.0
MOVL C07507 V=8.0
MOVL C07508 V=8.0
MOVL C07509 V=8.0
MOVL C07510 V=8.0
MOVL C07511 V=8.0
MOVL C07512 V=8.0
MOVL C07513 V=8.0
MOVL C07514 V=8.0
MOVL C07515 V=8.0
MOVL C07516 V=8.0
MOVL C07517 V=8.0
MOVL C07518 V=8.0
MOVL C07519 V=8.0
MOVL C07520 V=8.0
MOVL C07521 V=8.0
MOVL C07522 V=8.0
MOVL C07523 V=8.0
MOVJ C07524 VJ=0.78
MOVJ C07525 VJ=0.78
MOVL C07526 V=11.7
TIMER T=2.00
MOVL C07527 V=11.7
MOVJ C07528 VJ=0.78
MOVJ C07529 VJ=0.78
MOVL C07530 V=8.0
MOVL C07531 V=8.0
MOVL C07532 V=8.0
MOVL C07533 V=8.0
MOVL C07534 V=8.0
MOVL C07535 V=8.0
MOVL C07536 V=8.0
MOVL C07537 V=8.0
MOVL C07538 V=8.0
MOVL C07539 V=8.0
MOVL C07540 V=8.0
MOVL C07541 V=8.0
MOVL C07542 V=8.0
MOVL C07543 V=8.0
MOVL C07544 V=8.0
MOVL C07545 V=8.0
MOVL C07546 V=8.0
MOVL C07547 V=8.0
MOVL C07548 V=8.0
MOVL C07549 V=8.0
MOVL C07550 V=8.0
MOVL C07551 V=8.0
MOVJ C07552 VJ=0.78
MOVL C07553 V=8.0
MOVL C07554 V=8.0
MOVL C07555 V=8.0
MOVL C07556 V=8.0
MOVL C07557 V=8.0
MOVL C07558 V=8.0
MOVL C07559 V=8.0
MOVL C07560 V=8.0
MOVL C07561 V=8.0
MOVL C07562 V=8.0
MOVL C07563 V=8.0
MOVL C07564 V=8.0
MOVL C07565 V=8.0
MOVL C07566 V=8.0
MOVL C07567 V=8.0
MOVL C07568 V=8.0
MOVL C07569 V=8.0
MOVL C07570 V=8.0
MOVL C07571 V=8.0
MOVL C07572 V=8.0
MOVL C07573 V=8.0
MOVL C07574 V=8.0
MOVL C07575 V=8.0
MOVL C07576 V=8.0
MOVL C07577 V=8.0
MOVL C07578 V=8.0
MOVL C07579 V=8.0
MOVL C07580 V=8.0
MOVL C07581 V=8.0
MOVL C07582 V=8.0
MOVL C07583 V=8.0
MOVL C07584 V=8.0
MOVL C07585 V=8.0
MOVL C07586 V=8.0
MOVL C07587 V=8.0
MOVL C07588 V=8.0
MOVL C07589 V=8.0
MOVL C07590 V=8.0
MOVL C07591 V=8.0
MOVL C07592 V=8.0
MOVL C07593 V=8.0
MOVL C07594 V=8.0
MOVL C07595 V=8.0
MOVL C07596 V=8.0
MOVL C07597 V=8.0
MOVL C07598 V=8.0
MOVL C07599 V=8.0
MOVL C07600 V=8.0
MOVL C07601 V=8.0
MOVL C07602 V=8.0
MOVL C07603 V=8.0
MOVL C07604 V=8.0
MOVL C07605 V=8.0
MOVL C07606 V=8.0
MOVL C07607 V=8.0
MOVL C07608 V=8.0
MOVL C07609 V=8.0
MOVL C07610 V=8.0
MOVL C07611 V=8.0
MOVL C07612 V=8.0
MOVL C07613 V=8.0
MOVL C07614 V=8.0
MOVJ C07615 VJ=0.78
MOVL C07616 V=8.0
MOVL C07617 V=8.0
MOVL C07618 V=8.0
MOVL C07619 V=8.0
MOVL C07620 V=8.0
MOVL C07621 V=8.0
MOVL C07622 V=8.0
MOVL C07623 V=8.0
MOVL C07624 V=8.0
MOVL C07625 V=8.0
MOVL C07626 V=8.0
MOVL C07627 V=8.0
MOVL C07628 V=8.0
MOVL C07629 V=8.0
MOVL C07630 V=8.0
MOVL C07631 V=8.0
MOVL C07632 V=8.0
MOVL C07633 V=8.0
MOVL C07634 V=8.0
MOVL C07635 V=8.0
MOVL C07636 V=8.0
MOVL C07637 V=8.0
MOVL C07638 V=8.0
MOVL C07639 V=8.0
MOVL C07640 V=8.0
MOVL C07641 V=8.0
MOVL C07642 V=8.0
MOVL C07643 V=8.0
MOVL C07644 V=8.0
MOVL C07645 V=8.0
MOVL C07646 V=8.0
MOVL C07647 V=8.0
MOVL C07648 V=8.0
MOVL C07649 V=8.0
MOVL C07650 V=8.0
MOVL C07651 V=8.0
MOVL C07652 V=8.0
MOVL C07653 V=8.0
MOVL C07654 V=8.0
MOVL C07655 V=8.0
MOVL C07656 V=8.0
MOVL C07657 V=8.0
MOVL C07658 V=8.0
MOVL C07659 V=8.0
MOVL C07660 V=8.0
MOVL C07661 V=8.0
MOVL C07662 V=8.0
MOVL C07663 V=8.0
MOVL C07664 V=8.0
MOVL C07665 V=8.0
MOVL C07666 V=8.0
MOVL C07667 V=8.0
MOVL C07668 V=8.0
MOVL C07669 V=8.0
MOVL C07670 V=8.0
MOVL C07671 V=8.0
MOVL C07672 V=8.0
MOVL C07673 V=8.0
MOVL C07674 V=8.0
MOVL C07675 V=8.0
MOVL C07676 V=8.0
MOVL C07677 V=8.0
MOVJ C07678 VJ=0.78
MOVL C07679 V=8.0
MOVL C07680 V=8.0
MOVL C07681 V=8.0
MOVL C07682 V=8.0
MOVL C07683 V=8.0
MOVL C07684 V=8.0
MOVL C07685 V=8.0
MOVL C07686 V=8.0
MOVL C07687 V=8.0
MOVL C07688 V=8.0
MOVL C07689 V=8.0
MOVL C07690 V=8.0
MOVL C07691 V=8.0
MOVL C07692 V=8.0
MOVL C07693 V=8.0
MOVL C07694 V=8.0
MOVL C07695 V=8.0
MOVL C07696 V=8.0
MOVL C07697 V=8.0
MOVL C07698 V=8.0
MOVL C07699 V=8.0
MOVJ C07700 VJ=0.78
MOVJ C07701 VJ=0.78
MOVL C07702 V=11.7
TIMER T=2.00
MOVL C07703 V=11.7
MOVJ C07704 VJ=0.78
MOVJ C07705 VJ=0.78
MOVL C07706 V=8.0
MOVL C07707 V=8.0
MOVL C07708 V=8.0
MOVL C07709 V=8.0
MOVL C07710 V=8.0
MOVL C07711 V=8.0
MOVL C07712 V=8.0
MOVL C07713 V=8.0
MOVL C07714 V=8.0
MOVL C07715 V=8.0
MOVL C07716 V=8.0
MOVL C07717 V=8.0
MOVL C07718 V=8.0
MOVL C07719 V=8.0
MOVL C07720 V=8.0
MOVL C07721 V=8.0
MOVL C07722 V=8.0
MOVL C07723 V=8.0
MOVL C07724 V=8.0
MOVL C07725 V=8.0
MOVL C07726 V=8.0
MOVL C07727 V=8.0
MOVL C07728 V=8.0
MOVL C07729 V=8.0
MOVL C07730 V=8.0
MOVL C07731 V=8.0
MOVL C07732 V=8.0
MOVL C07733 V=8.0
MOVL C07734 V=8.0
MOVL C07735 V=8.0
MOVL C07736 V=8.0
MOVL C07737 V=8.0
MOVL C07738 V=8.0
MOVL C07739 V=8.0
MOVL C07740 V=8.0
MOVL C07741 V=8.0
MOVL C07742 V=8.0
MOVL C07743 V=8.0
MOVL C07744 V=8.0
MOVL C07745 V=8.0
MOVL C07746 V=8.0
MOVL C07747 V=8.0
MOVJ C07748 VJ=0.78
MOVL C07749 V=8.0
MOVL C07750 V=8.0
MOVL C07751 V=8.0
MOVL C07752 V=8.0
MOVL C07753 V=8.0
MOVL C07754 V=8.0
MOVL C07755 V=8.0
MOVL C07756 V=8.0
MOVL C07757 V=8.0
MOVL C07758 V=8.0
MOVL C07759 V=8.0
MOVL C07760 V=8.0
MOVL C07761 V=8.0
MOVL C07762 V=8.0
MOVL C07763 V=8.0
MOVL C07764 V=8.0
MOVL C07765 V=8.0
MOVL C07766 V=8.0
MOVL C07767 V=8.0
MOVL C07768 V=8.0
MOVL C07769 V=8.0
MOVL C07770 V=8.0
MOVL C07771 V=8.0
MOVL C07772 V=8.0
MOVL C07773 V=8.0
MOVL C07774 V=8.0
MOVL C07775 V=8.0
MOVL C07776 V=8.0
MOVL C07777 V=8.0
MOVL C07778 V=8.0
MOVL C07779 V=8.0
MOVL C07780 V=8.0
MOVL C07781 V=8.0
MOVL C07782 V=8.0
MOVL C07783 V=8.0
MOVL C07784 V=8.0
MOVL C07785 V=8.0
MOVL C07786 V=8.0
MOVL C07787 V=8.0
MOVL C07788 V=8.0
MOVL C07789 V=8.0
MOVL C07790 V=8.0
MOVL C07791 V=8.0
MOVL C07792 V=8.0
MOVL C07793 V=8.0
MOVL C07794 V=8.0
MOVL C07795 V=8.0
MOVL C07796 V=8.0
MOVL C07797 V=8.0
MOVL C07798 V=8.0
MOVL C07799 V=8.0
MOVL C07800 V=8.0
MOVL C07801 V=8.0
MOVL C07802 V=8.0
MOVL C07803 V=8.0
MOVL C07804 V=8.0
MOVL C07805 V=8.0
MOVL C07806 V=8.0
MOVL C07807 V=8.0
MOVL C07808 V=8.0
MOVL C07809 V=8.0
MOVL C07810 V=8.0
MOVJ C07811 VJ=0.78
MOVL C07812 V=8.0
MOVL C07813 V=8.0
MOVL C07814 V=8.0
MOVL C07815 V=8.0
MOVL C07816 V=8.0
MOVL C07817 V=8.0
MOVL C07818 V=8.0
MOVL C07819 V=8.0
MOVL C07820 V=8.0
MOVL C07821 V=8.0
MOVL C07822 V=8.0
MOVL C07823 V=8.0
MOVL C07824 V=8.0
MOVL C07825 V=8.0
MOVL C07826 V=8.0
MOVL C07827 V=8.0
MOVL C07828 V=8.0
MOVL C07829 V=8.0
MOVL C07830 V=8.0
MOVL C07831 V=8.0
MOVL C07832 V=8.0
MOVL C07833 V=8.0
MOVL C07834 V=8.0
MOVL C07835 V=8.0
MOVL C07836 V=8.0
MOVL C07837 V=8.0
MOVL C07838 V=8.0
MOVL C07839 V=8.0
MOVL C07840 V=8.0
MOVL C07841 V=8.0
MOVL C07842 V=8.0
MOVL C07843 V=8.0
MOVL C07844 V=8.0
MOVL C07845 V=8.0
MOVL C07846 V=8.0
MOVL C07847 V=8.0
MOVL C07848 V=8.0
MOVL C07849 V=8.0
MOVL C07850 V=8.0
MOVL C07851 V=8.0
MOVL C07852 V=8.0
MOVL C07853 V=8.0
MOVL C07854 V=8.0
MOVL C07855 V=8.0
MOVL C07856 V=8.0
MOVL C07857 V=8.0
MOVL C07858 V=8.0
MOVL C07859 V=8.0
MOVL C07860 V=8.0
MOVL C07861 V=8.0
MOVL C07862 V=8.0
MOVL C07863 V=8.0
MOVL C07864 V=8.0
MOVL C07865 V=8.0
MOVL C07866 V=8.0
MOVL C07867 V=8.0
MOVL C07868 V=8.0
MOVL C07869 V=8.0
MOVL C07870 V=8.0
MOVL C07871 V=8.0
MOVL C07872 V=8.0
MOVJ C07873 VJ=0.78
MOVJ C07874 VJ=0.78
MOVL C07875 V=11.7
TIMER T=2.00
MOVL C07876 V=11.7
MOVJ C07877 VJ=0.78
MOVJ C07878 VJ=0.78
MOVL C07879 V=8.0
MOVL C07880 V=8.0
MOVJ C07881 VJ=0.78
MOVL C07882 V=8.0
MOVL C07883 V=8.0
MOVL C07884 V=8.0
MOVL C07885 V=8.0
MOVL C07886 V=8.0
MOVL C07887 V=8.0
MOVL C07888 V=8.0
MOVL C07889 V=8.0
MOVL C07890 V=8.0
MOVL C07891 V=8.0
MOVL C07892 V=8.0
MOVL C07893 V=8.0
MOVL C07894 V=8.0
MOVL C07895 V=8.0
MOVL C07896 V=8.0
MOVL C07897 V=8.0
MOVL C07898 V=8.0
MOVL C07899 V=8.0
MOVL C07900 V=8.0
MOVL C07901 V=8.0
MOVL C07902 V=8.0
MOVL C07903 V=8.0
MOVL C07904 V=8.0
MOVL C07905 V=8.0
MOVL C07906 V=8.0
MOVL C07907 V=8.0
MOVL C07908 V=8.0
MOVL C07909 V=8.0
MOVL C07910 V=8.0
MOVL C07911 V=8.0
MOVL C07912 V=8.0
MOVL C07913 V=8.0
MOVL C07914 V=8.0
MOVL C07915 V=8.0
MOVL C07916 V=8.0
MOVL C07917 V=8.0
MOVL C07918 V=8.0
MOVL C07919 V=8.0
MOVL C07920 V=8.0
MOVL C07921 V=8.0
MOVL C07922 V=8.0
MOVL C07923 V=8.0
MOVL C07924 V=8.0
MOVL C07925 V=8.0
MOVL C07926 V=8.0
MOVL C07927 V=8.0
MOVL C07928 V=8.0
MOVL C07929 V=8.0
MOVL C07930 V=8.0
MOVL C07931 V=8.0
MOVL C07932 V=8.0
MOVL C07933 V=8.0
MOVL C07934 V=8.0
MOVL C07935 V=8.0
MOVL C07936 V=8.0
MOVL C07937 V=8.0
MOVL C07938 V=8.0
MOVL C07939 V=8.0
MOVL C07940 V=8.0
MOVL C07941 V=8.0
MOVL C07942 V=8.0
MOVL C07943 V=8.0
MOVJ C07944 VJ=0.78
MOVL C07945 V=8.0
MOVL C07946 V=8.0
MOVL C07947 V=8.0
MOVL C07948 V=8.0
MOVL C07949 V=8.0
MOVL C07950 V=8.0
MOVL C07951 V=8.0
MOVL C07952 V=8.0
MOVL C07953 V=8.0
MOVL C07954 V=8.0
MOVL C07955 V=8.0
MOVL C07956 V=8.0
MOVL C07957 V=8.0
MOVL C07958 V=8.0
MOVL C07959 V=8.0
MOVL C07960 V=8.0
MOVL C07961 V=8.0
MOVL C07962 V=8.0
MOVL C07963 V=8.0
MOVL C07964 V=8.0
MOVL C07965 V=8.0
MOVL C07966 V=8.0
MOVL C07967 V=8.0
MOVL C07968 V=8.0
MOVL C07969 V=8.0
MOVL C07970 V=8.0
MOVL C07971 V=8.0
MOVL C07972 V=8.0
MOVL C07973 V=8.0
MOVL C07974 V=8.0
MOVL C07975 V=8.0
MOVL C07976 V=8.0
MOVL C07977 V=8.0
MOVL C07978 V=8.0
MOVL C07979 V=8.0
MOVL C07980 V=8.0
MOVL C07981 V=8.0
MOVL C07982 V=8.0
MOVL C07983 V=8.0
MOVL C07984 V=8.0
MOVL C07985 V=8.0
MOVL C07986 V=8.0
MOVL C07987 V=8.0
MOVL C07988 V=8.0
MOVL C07989 V=8.0
MOVL C07990 V=8.0
MOVL C07991 V=8.0
MOVL C07992 V=8.0
MOVL C07993 V=8.0
MOVL C07994 V=8.0
MOVL C07995 V=8.0
MOVL C07996 V=8.0
MOVL C07997 V=8.0
MOVL C07998 V=8.0
MOVL C07999 V=8.0
MOVL C08000 V=8.0
MOVL C08001 V=8.0
MOVL C08002 V=8.0
MOVL C08003 V=8.0
MOVL C08004 V=8.0
MOVL C08005 V=8.0
MOVL C08006 V=8.0
MOVJ C08007 VJ=0.78
MOVL C08008 V=8.0
MOVL C08009 V=8.0
MOVL C08010 V=8.0
MOVL C08011 V=8.0
MOVL C08012 V=8.0
MOVL C08013 V=8.0
MOVL C08014 V=8.0
MOVL C08015 V=8.0
MOVL C08016 V=8.0
MOVL C08017 V=8.0
MOVL C08018 V=8.0
MOVL C08019 V=8.0
MOVL C08020 V=8.0
MOVL C08021 V=8.0
MOVL C08022 V=8.0
MOVL C08023 V=8.0
MOVL C08024 V=8.0
MOVL C08025 V=8.0
MOVL C08026 V=8.0
MOVL C08027 V=8.0
MOVL C08028 V=8.0
MOVL C08029 V=8.0
MOVL C08030 V=8.0
MOVL C08031 V=8.0
MOVL C08032 V=8.0
MOVL C08033 V=8.0
MOVL C08034 V=8.0
MOVL C08035 V=8.0
MOVL C08036 V=8.0
MOVL C08037 V=8.0
MOVL C08038 V=8.0
MOVL C08039 V=8.0
MOVL C08040 V=8.0
MOVL C08041 V=8.0
MOVL C08042 V=8.0
MOVL C08043 V=8.0
MOVL C08044 V=8.0
MOVL C08045 V=8.0
MOVL C08046 V=8.0
MOVL C08047 V=8.0
MOVL C08048 V=8.0
MOVJ C08049 VJ=0.78
MOVJ C08050 VJ=0.78
MOVL C08051 V=11.7
TIMER T=2.00
MOVL C08052 V=11.7
MOVJ C08053 VJ=0.78
MOVJ C08054 VJ=0.78
MOVL C08055 V=8.0
MOVL C08056 V=8.0
MOVL C08057 V=8.0
MOVL C08058 V=8.0
MOVL C08059 V=8.0
MOVL C08060 V=8.0
MOVL C08061 V=8.0
MOVL C08062 V=8.0
MOVL C08063 V=8.0
MOVL C08064 V=8.0
MOVL C08065 V=8.0
MOVL C08066 V=8.0
MOVL C08067 V=8.0
MOVL C08068 V=8.0
MOVL C08069 V=8.0
MOVL C08070 V=8.0
MOVL C08071 V=8.0
MOVL C08072 V=8.0
MOVL C08073 V=8.0
MOVL C08074 V=8.0
MOVL C08075 V=8.0
MOVL C08076 V=8.0
MOVJ C08077 VJ=0.78
MOVL C08078 V=8.0
MOVL C08079 V=8.0
MOVL C08080 V=8.0
MOVL C08081 V=8.0
MOVL C08082 V=8.0
MOVL C08083 V=8.0
MOVL C08084 V=8.0
MOVL C08085 V=8.0
MOVL C08086 V=8.0
MOVL C08087 V=8.0
MOVL C08088 V=8.0
MOVL C08089 V=8.0
MOVL C08090 V=8.0
MOVL C08091 V=8.0
MOVL C08092 V=8.0
MOVL C08093 V=8.0
MOVL C08094 V=8.0
MOVL C08095 V=8.0
MOVL C08096 V=8.0
MOVL C08097 V=8.0
MOVL C08098 V=8.0
MOVL C08099 V=8.0
MOVL C08100 V=8.0
MOVL C08101 V=8.0
MOVL C08102 V=8.0
MOVL C08103 V=8.0
MOVL C08104 V=8.0
MOVL C08105 V=8.0
MOVL C08106 V=8.0
MOVL C08107 V=8.0
MOVL C08108 V=8.0
MOVL C08109 V=8.0
MOVL C08110 V=8.0
MOVL C08111 V=8.0
MOVL C08112 V=8.0
MOVL C08113 V=8.0
MOVL C08114 V=8.0
MOVL C08115 V=8.0
MOVL C08116 V=8.0
MOVL C08117 V=8.0
MOVL C08118 V=8.0
MOVL C08119 V=8.0
MOVL C08120 V=8.0
MOVL C08121 V=8.0
MOVL C08122 V=8.0
MOVL C08123 V=8.0
MOVL C08124 V=8.0
MOVL C08125 V=8.0
MOVL C08126 V=8.0
MOVL C08127 V=8.0
MOVL C08128 V=8.0
MOVL C08129 V=8.0
MOVL C08130 V=8.0
MOVL C08131 V=8.0
MOVL C08132 V=8.0
MOVL C08133 V=8.0
MOVL C08134 V=8.0
MOVL C08135 V=8.0
MOVL C08136 V=8.0
MOVL C08137 V=8.0
MOVL C08138 V=8.0
MOVL C08139 V=8.0
MOVJ C08140 VJ=0.78
MOVL C08141 V=8.0
MOVL C08142 V=8.0
MOVL C08143 V=8.0
MOVL C08144 V=8.0
MOVL C08145 V=8.0
MOVL C08146 V=8.0
MOVL C08147 V=8.0
MOVL C08148 V=8.0
MOVL C08149 V=8.0
MOVL C08150 V=8.0
MOVL C08151 V=8.0
MOVL C08152 V=8.0
MOVL C08153 V=8.0
MOVL C08154 V=8.0
MOVL C08155 V=8.0
MOVL C08156 V=8.0
MOVL C08157 V=8.0
MOVL C08158 V=8.0
MOVL C08159 V=8.0
MOVL C08160 V=8.0
MOVL C08161 V=8.0
MOVL C08162 V=8.0
MOVL C08163 V=8.0
MOVL C08164 V=8.0
MOVL C08165 V=8.0
MOVL C08166 V=8.0
MOVL C08167 V=8.0
MOVL C08168 V=8.0
MOVL C08169 V=8.0
MOVL C08170 V=8.0
MOVL C08171 V=8.0
MOVL C08172 V=8.0
MOVL C08173 V=8.0
MOVL C08174 V=8.0
MOVL C08175 V=8.0
MOVL C08176 V=8.0
MOVL C08177 V=8.0
MOVL C08178 V=8.0
MOVL C08179 V=8.0
MOVL C08180 V=8.0
MOVL C08181 V=8.0
MOVL C08182 V=8.0
MOVL C08183 V=8.0
MOVL C08184 V=8.0
MOVL C08185 V=8.0
MOVL C08186 V=8.0
MOVL C08187 V=8.0
MOVL C08188 V=8.0
MOVL C08189 V=8.0
MOVL C08190 V=8.0
MOVL C08191 V=8.0
MOVL C08192 V=8.0
MOVL C08193 V=8.0
MOVL C08194 V=8.0
MOVL C08195 V=8.0
MOVL C08196 V=8.0
MOVL C08197 V=8.0
MOVL C08198 V=8.0
MOVL C08199 V=8.0
MOVL C08200 V=8.0
MOVL C08201 V=8.0
MOVL C08202 V=8.0
MOVJ C08203 VJ=0.78
MOVL C08204 V=8.0
MOVL C08205 V=8.0
MOVL C08206 V=8.0
MOVL C08207 V=8.0
MOVL C08208 V=8.0
MOVL C08209 V=8.0
MOVL C08210 V=8.0
MOVL C08211 V=8.0
MOVL C08212 V=8.0
MOVL C08213 V=8.0
MOVL C08214 V=8.0
MOVL C08215 V=8.0
MOVL C08216 V=8.0
MOVL C08217 V=8.0
MOVL C08218 V=8.0
MOVL C08219 V=8.0
MOVL C08220 V=8.0
MOVL C08221 V=8.0
MOVL C08222 V=8.0
MOVL C08223 V=8.0
MOVL C08224 V=8.0
MOVJ C08225 VJ=0.78
MOVJ C08226 VJ=0.78
MOVL C08227 V=11.7
TIMER T=2.00
MOVL C08228 V=11.7
MOVJ C08229 VJ=0.78
MOVJ C08230 VJ=0.78
MOVL C08231 V=8.0
MOVL C08232 V=8.0
MOVL C08233 V=8.0
MOVL C08234 V=8.0
MOVL C08235 V=8.0
MOVL C08236 V=8.0
MOVL C08237 V=8.0
MOVL C08238 V=8.0
MOVL C08239 V=8.0
MOVL C08240 V=8.0
MOVL C08241 V=8.0
MOVL C08242 V=8.0
MOVL C08243 V=8.0
MOVL C08244 V=8.0
MOVL C08245 V=8.0
MOVL C08246 V=8.0
MOVL C08247 V=8.0
MOVL C08248 V=8.0
MOVL C08249 V=8.0
MOVL C08250 V=8.0
MOVL C08251 V=8.0
MOVL C08252 V=8.0
MOVL C08253 V=8.0
MOVL C08254 V=8.0
MOVL C08255 V=8.0
MOVL C08256 V=8.0
MOVL C08257 V=8.0
MOVL C08258 V=8.0
MOVL C08259 V=8.0
MOVL C08260 V=8.0
MOVL C08261 V=8.0
MOVL C08262 V=8.0
MOVL C08263 V=8.0
MOVL C08264 V=8.0
MOVL C08265 V=8.0
MOVL C08266 V=8.0
MOVL C08267 V=8.0
MOVL C08268 V=8.0
MOVL C08269 V=8.0
MOVL C08270 V=8.0
MOVL C08271 V=8.0
MOVL C08272 V=8.0
MOVJ C08273 VJ=0.78
MOVL C08274 V=8.0
MOVL C08275 V=8.0
MOVL C08276 V=8.0
MOVL C08277 V=8.0
MOVL C08278 V=8.0
MOVL C08279 V=8.0
MOVL C08280 V=8.0
MOVL C08281 V=8.0
MOVL C08282 V=8.0
MOVL C08283 V=8.0
MOVL C08284 V=8.0
MOVL C08285 V=8.0
MOVL C08286 V=8.0
MOVL C08287 V=8.0
MOVL C08288 V=8.0
MOVL C08289 V=8.0
MOVL C08290 V=8.0
MOVL C08291 V=8.0
MOVL C08292 V=8.0
MOVL C08293 V=8.0
MOVL C08294 V=8.0
MOVL C08295 V=8.0
MOVL C08296 V=8.0
MOVL C08297 V=8.0
MOVL C08298 V=8.0
MOVL C08299 V=8.0
MOVL C08300 V=8.0
MOVL C08301 V=8.0
MOVL C08302 V=8.0
MOVL C08303 V=8.0
MOVL C08304 V=8.0
MOVL C08305 V=8.0
MOVL C08306 V=8.0
MOVL C08307 V=8.0
MOVL C08308 V=8.0
MOVL C08309 V=8.0
MOVL C08310 V=8.0
MOVL C08311 V=8.0
MOVL C08312 V=8.0
MOVL C08313 V=8.0
MOVL C08314 V=8.0
MOVL C08315 V=8.0
MOVL C08316 V=8.0
MOVL C08317 V=8.0
MOVL C08318 V=8.0
MOVL C08319 V=8.0
MOVL C08320 V=8.0
MOVL C08321 V=8.0
MOVL C08322 V=8.0
MOVL C08323 V=8.0
MOVL C08324 V=8.0
MOVL C08325 V=8.0
MOVL C08326 V=8.0
MOVL C08327 V=8.0
MOVL C08328 V=8.0
MOVL C08329 V=8.0
MOVL C08330 V=8.0
MOVL C08331 V=8.0
MOVL C08332 V=8.0
MOVL C08333 V=8.0
MOVL C08334 V=8.0
MOVL C08335 V=8.0
MOVJ C08336 VJ=0.78
MOVL C08337 V=8.0
MOVL C08338 V=8.0
MOVL C08339 V=8.0
MOVL C08340 V=8.0
MOVL C08341 V=8.0
MOVL C08342 V=8.0
MOVL C08343 V=8.0
MOVL C08344 V=8.0
MOVL C08345 V=8.0
MOVL C08346 V=8.0
MOVL C08347 V=8.0
MOVL C08348 V=8.0
MOVL C08349 V=8.0
MOVL C08350 V=8.0
MOVL C08351 V=8.0
MOVL C08352 V=8.0
MOVL C08353 V=8.0
MOVL C08354 V=8.0
MOVL C08355 V=8.0
MOVL C08356 V=8.0
MOVL C08357 V=8.0
MOVL C08358 V=8.0
MOVL C08359 V=8.0
MOVL C08360 V=8.0
MOVL C08361 V=8.0
MOVL C08362 V=8.0
MOVL C08363 V=8.0
MOVL C08364 V=8.0
MOVL C08365 V=8.0
MOVL C08366 V=8.0
MOVL C08367 V=8.0
MOVL C08368 V=8.0
MOVL C08369 V=8.0
MOVL C08370 V=8.0
MOVL C08371 V=8.0
MOVL C08372 V=8.0
MOVL C08373 V=8.0
MOVL C08374 V=8.0
MOVL C08375 V=8.0
MOVL C08376 V=8.0
MOVL C08377 V=8.0
MOVL C08378 V=8.0
MOVL C08379 V=8.0
MOVL C08380 V=8.0
MOVL C08381 V=8.0
MOVL C08382 V=8.0
MOVL C08383 V=8.0
MOVL C08384 V=8.0
MOVL C08385 V=8.0
MOVL C08386 V=8.0
MOVL C08387 V=8.0
MOVL C08388 V=8.0
MOVL C08389 V=8.0
MOVL C08390 V=8.0
MOVL C08391 V=8.0
MOVL C08392 V=8.0
MOVL C08393 V=8.0
MOVL C08394 V=8.0
MOVL C08395 V=8.0
MOVL C08396 V=8.0
MOVL C08397 V=8.0
MOVJ C08398 VJ=0.78
MOVJ C08399 VJ=0.78
MOVL C08400 V=11.7
TIMER T=2.00
MOVL C08401 V=11.7
MOVJ C08402 VJ=0.78
MOVJ C08403 VJ=0.78
MOVL C08404 V=8.0
MOVL C08405 V=8.0
MOVJ C08406 VJ=0.78
MOVL C08407 V=8.0
MOVL C08408 V=8.0
MOVL C08409 V=8.0
MOVL C08410 V=8.0
MOVL C08411 V=8.0
MOVL C08412 V=8.0
MOVL C08413 V=8.0
MOVL C08414 V=8.0
MOVL C08415 V=8.0
MOVL C08416 V=8.0
MOVL C08417 V=8.0
MOVL C08418 V=8.0
MOVL C08419 V=8.0
MOVL C08420 V=8.0
MOVL C08421 V=8.0
MOVL C08422 V=8.0
MOVL C08423 V=8.0
MOVL C08424 V=8.0
MOVL C08425 V=8.0
MOVL C08426 V=8.0
MOVL C08427 V=8.0
MOVL C08428 V=8.0
MOVL C08429 V=8.0
MOVL C08430 V=8.0
MOVL C08431 V=8.0
MOVL C08432 V=8.0
MOVL C08433 V=8.0
MOVL C08434 V=8.0
MOVL C08435 V=8.0
MOVL C08436 V=8.0
MOVL C08437 V=8.0
MOVL C08438 V=8.0
MOVL C08439 V=8.0
MOVL C08440 V=8.0
MOVL C08441 V=8.0
MOVL C08442 V=8.0
MOVL C08443 V=8.0
MOVL C08444 V=8.0
MOVL C08445 V=8.0
MOVL C08446 V=8.0
MOVL C08447 V=8.0
MOVL C08448 V=8.0
MOVL C08449 V=8.0
MOVL C08450 V=8.0
MOVL C08451 V=8.0
MOVL C08452 V=8.0
MOVL C08453 V=8.0
MOVL C08454 V=8.0
MOVL C08455 V=8.0
MOVL C08456 V=8.0
MOVL C08457 V=8.0
MOVL C08458 V=8.0
MOVL C08459 V=8.0
MOVL C08460 V=8.0
MOVL C08461 V=8.0
MOVL C08462 V=8.0
MOVL C08463 V=8.0
MOVL C08464 V=8.0
MOVL C08465 V=8.0
MOVL C08466 V=8.0
MOVL C08467 V=8.0
MOVL C08468 V=8.0
MOVJ C08469 VJ=0.78
MOVL C08470 V=8.0
MOVL C08471 V=8.0
MOVL C08472 V=8.0
MOVL C08473 V=8.0
MOVL C08474 V=8.0
MOVL C08475 V=8.0
MOVL C08476 V=8.0
MOVL C08477 V=8.0
MOVL C08478 V=8.0
MOVL C08479 V=8.0
MOVL C08480 V=8.0
MOVL C08481 V=8.0
MOVL C08482 V=8.0
MOVL C08483 V=8.0
MOVL C08484 V=8.0
MOVL C08485 V=8.0
MOVL C08486 V=8.0
MOVL C08487 V=8.0
MOVL C08488 V=8.0
MOVL C08489 V=8.0
MOVL C08490 V=8.0
MOVL C08491 V=8.0
MOVL C08492 V=8.0
MOVL C08493 V=8.0
MOVL C08494 V=8.0
MOVL C08495 V=8.0
MOVL C08496 V=8.0
MOVL C08497 V=8.0
MOVL C08498 V=8.0
MOVL C08499 V=8.0
MOVL C08500 V=8.0
MOVL C08501 V=8.0
MOVL C08502 V=8.0
MOVL C08503 V=8.0
MOVL C08504 V=8.0
MOVL C08505 V=8.0
MOVL C08506 V=8.0
MOVL C08507 V=8.0
MOVL C08508 V=8.0
MOVL C08509 V=8.0
MOVL C08510 V=8.0
MOVL C08511 V=8.0
MOVL C08512 V=8.0
MOVL C08513 V=8.0
MOVL C08514 V=8.0
MOVL C08515 V=8.0
MOVL C08516 V=8.0
MOVL C08517 V=8.0
MOVL C08518 V=8.0
MOVL C08519 V=8.0
MOVL C08520 V=8.0
MOVL C08521 V=8.0
MOVL C08522 V=8.0
MOVL C08523 V=8.0
MOVL C08524 V=8.0
MOVL C08525 V=8.0
MOVL C08526 V=8.0
MOVL C08527 V=8.0
MOVL C08528 V=8.0
MOVL C08529 V=8.0
MOVL C08530 V=8.0
MOVL C08531 V=8.0
MOVJ C08532 VJ=0.78
MOVL C08533 V=8.0
MOVL C08534 V=8.0
MOVL C08535 V=8.0
MOVL C08536 V=8.0
MOVL C08537 V=8.0
MOVL C08538 V=8.0
MOVL C08539 V=8.0
MOVL C08540 V=8.0
MOVL C08541 V=8.0
MOVL C08542 V=8.0
MOVL C08543 V=8.0
MOVL C08544 V=8.0
MOVL C08545 V=8.0
MOVL C08546 V=8.0
MOVL C08547 V=8.0
MOVL C08548 V=8.0
MOVL C08549 V=8.0
MOVL C08550 V=8.0
MOVL C08551 V=8.0
MOVL C08552 V=8.0
MOVL C08553 V=8.0
MOVL C08554 V=8.0
MOVL C08555 V=8.0
MOVL C08556 V=8.0
MOVL C08557 V=8.0
MOVL C08558 V=8.0
MOVL C08559 V=8.0
MOVL C08560 V=8.0
MOVL C08561 V=8.0
MOVL C08562 V=8.0
MOVL C08563 V=8.0
MOVL C08564 V=8.0
MOVL C08565 V=8.0
MOVL C08566 V=8.0
MOVL C08567 V=8.0
MOVL C08568 V=8.0
MOVL C08569 V=8.0
MOVL C08570 V=8.0
MOVL C08571 V=8.0
MOVL C08572 V=8.0
MOVL C08573 V=8.0
MOVJ C08574 VJ=0.78
MOVJ C08575 VJ=0.78
MOVL C08576 V=11.7
TIMER T=2.00
MOVL C08577 V=11.7
MOVJ C08578 VJ=0.78
MOVJ C08579 VJ=0.78
MOVL C08580 V=8.0
MOVL C08581 V=8.0
MOVL C08582 V=8.0
MOVL C08583 V=8.0
MOVL C08584 V=8.0
MOVL C08585 V=8.0
MOVL C08586 V=8.0
MOVL C08587 V=8.0
MOVL C08588 V=8.0
MOVL C08589 V=8.0
MOVL C08590 V=8.0
MOVL C08591 V=8.0
MOVL C08592 V=8.0
MOVL C08593 V=8.0
MOVL C08594 V=8.0
MOVL C08595 V=8.0
MOVL C08596 V=8.0
MOVL C08597 V=8.0
MOVL C08598 V=8.0
MOVL C08599 V=8.0
MOVL C08600 V=8.0
MOVL C08601 V=8.0
MOVJ C08602 VJ=0.78
MOVL C08603 V=8.0
MOVL C08604 V=8.0
MOVL C08605 V=8.0
MOVL C08606 V=8.0
MOVL C08607 V=8.0
MOVL C08608 V=8.0
MOVL C08609 V=8.0
MOVL C08610 V=8.0
MOVL C08611 V=8.0
MOVL C08612 V=8.0
MOVL C08613 V=8.0
MOVL C08614 V=8.0
MOVL C08615 V=8.0
MOVL C08616 V=8.0
MOVL C08617 V=8.0
MOVL C08618 V=8.0
MOVL C08619 V=8.0
MOVL C08620 V=8.0
MOVL C08621 V=8.0
MOVL C08622 V=8.0
MOVL C08623 V=8.0
MOVL C08624 V=8.0
MOVL C08625 V=8.0
MOVL C08626 V=8.0
MOVL C08627 V=8.0
MOVL C08628 V=8.0
MOVL C08629 V=8.0
MOVL C08630 V=8.0
MOVL C08631 V=8.0
MOVL C08632 V=8.0
MOVL C08633 V=8.0
MOVL C08634 V=8.0
MOVL C08635 V=8.0
MOVL C08636 V=8.0
MOVL C08637 V=8.0
MOVL C08638 V=8.0
MOVL C08639 V=8.0
MOVL C08640 V=8.0
MOVL C08641 V=8.0
MOVL C08642 V=8.0
MOVL C08643 V=8.0
MOVL C08644 V=8.0
MOVL C08645 V=8.0
MOVL C08646 V=8.0
MOVL C08647 V=8.0
MOVL C08648 V=8.0
MOVL C08649 V=8.0
MOVL C08650 V=8.0
MOVL C08651 V=8.0
MOVL C08652 V=8.0
MOVL C08653 V=8.0
MOVL C08654 V=8.0
MOVL C08655 V=8.0
MOVL C08656 V=8.0
MOVL C08657 V=8.0
MOVL C08658 V=8.0
MOVL C08659 V=8.0
MOVL C08660 V=8.0
MOVL C08661 V=8.0
MOVL C08662 V=8.0
MOVL C08663 V=8.0
MOVL C08664 V=8.0
MOVJ C08665 VJ=0.78
MOVL C08666 V=8.0
MOVL C08667 V=8.0
MOVL C08668 V=8.0
MOVL C08669 V=8.0
MOVL C08670 V=8.0
MOVL C08671 V=8.0
MOVL C08672 V=8.0
MOVL C08673 V=8.0
MOVL C08674 V=8.0
MOVL C08675 V=8.0
MOVL C08676 V=8.0
MOVL C08677 V=8.0
MOVL C08678 V=8.0
MOVL C08679 V=8.0
MOVL C08680 V=8.0
MOVL C08681 V=8.0
MOVL C08682 V=8.0
MOVL C08683 V=8.0
MOVL C08684 V=8.0
MOVL C08685 V=8.0
MOVL C08686 V=8.0
MOVL C08687 V=8.0
MOVL C08688 V=8.0
MOVL C08689 V=8.0
MOVL C08690 V=8.0
MOVL C08691 V=8.0
MOVL C08692 V=8.0
MOVL C08693 V=8.0
MOVL C08694 V=8.0
MOVL C08695 V=8.0
MOVL C08696 V=8.0
MOVL C08697 V=8.0
MOVL C08698 V=8.0
MOVL C08699 V=8.0
MOVL C08700 V=8.0
MOVL C08701 V=8.0
MOVL C08702 V=8.0
MOVL C08703 V=8.0
MOVL C08704 V=8.0
MOVL C08705 V=8.0
MOVL C08706 V=8.0
MOVL C08707 V=8.0
MOVL C08708 V=8.0
MOVL C08709 V=8.0
MOVL C08710 V=8.0
MOVL C08711 V=8.0
MOVL C08712 V=8.0
MOVL C08713 V=8.0
MOVL C08714 V=8.0
MOVL C08715 V=8.0
MOVL C08716 V=8.0
MOVL C08717 V=8.0
MOVL C08718 V=8.0
MOVL C08719 V=8.0
MOVL C08720 V=8.0
MOVL C08721 V=8.0
MOVL C08722 V=8.0
MOVL C08723 V=8.0
MOVL C08724 V=8.0
MOVL C08725 V=8.0
MOVL C08726 V=8.0
MOVL C08727 V=8.0
MOVJ C08728 VJ=0.78
MOVL C08729 V=8.0
MOVL C08730 V=8.0
MOVL C08731 V=8.0
MOVL C08732 V=8.0
MOVL C08733 V=8.0
MOVL C08734 V=8.0
MOVL C08735 V=8.0
MOVL C08736 V=8.0
MOVL C08737 V=8.0
MOVL C08738 V=8.0
MOVL C08739 V=8.0
MOVL C08740 V=8.0
MOVL C08741 V=8.0
MOVL C08742 V=8.0
MOVL C08743 V=8.0
MOVL C08744 V=8.0
MOVL C08745 V=8.0
MOVL C08746 V=8.0
MOVL C08747 V=8.0
MOVL C08748 V=8.0
MOVL C08749 V=8.0
MOVJ C08750 VJ=0.78
MOVJ C08751 VJ=0.78
MOVL C08752 V=11.7
TIMER T=2.00
MOVL C08753 V=11.7
MOVJ C08754 VJ=0.78
MOVJ C08755 VJ=0.78
MOVL C08756 V=8.0
MOVL C08757 V=8.0
MOVL C08758 V=8.0
MOVL C08759 V=8.0
MOVL C08760 V=8.0
MOVL C08761 V=8.0
MOVL C08762 V=8.0
MOVL C08763 V=8.0
MOVL C08764 V=8.0
MOVL C08765 V=8.0
MOVL C08766 V=8.0
MOVL C08767 V=8.0
MOVL C08768 V=8.0
MOVL C08769 V=8.0
MOVL C08770 V=8.0
MOVL C08771 V=8.0
MOVL C08772 V=8.0
MOVL C08773 V=8.0
MOVL C08774 V=8.0
MOVL C08775 V=8.0
MOVL C08776 V=8.0
MOVL C08777 V=8.0
MOVL C08778 V=8.0
MOVL C08779 V=8.0
MOVL C08780 V=8.0
MOVL C08781 V=8.0
MOVL C08782 V=8.0
MOVL C08783 V=8.0
MOVL C08784 V=8.0
MOVL C08785 V=8.0
MOVL C08786 V=8.0
MOVL C08787 V=8.0
MOVL C08788 V=8.0
MOVL C08789 V=8.0
MOVL C08790 V=8.0
MOVL C08791 V=8.0
MOVL C08792 V=8.0
MOVL C08793 V=8.0
MOVL C08794 V=8.0
MOVL C08795 V=8.0
MOVL C08796 V=8.0
MOVL C08797 V=8.0
MOVJ C08798 VJ=0.78
MOVL C08799 V=8.0
MOVL C08800 V=8.0
MOVL C08801 V=8.0
MOVL C08802 V=8.0
MOVL C08803 V=8.0
MOVL C08804 V=8.0
MOVL C08805 V=8.0
MOVL C08806 V=8.0
MOVL C08807 V=8.0
MOVL C08808 V=8.0
MOVL C08809 V=8.0
MOVL C08810 V=8.0
MOVL C08811 V=8.0
MOVL C08812 V=8.0
MOVL C08813 V=8.0
MOVL C08814 V=8.0
MOVL C08815 V=8.0
MOVL C08816 V=8.0
MOVL C08817 V=8.0
MOVL C08818 V=8.0
MOVL C08819 V=8.0
MOVL C08820 V=8.0
MOVL C08821 V=8.0
MOVL C08822 V=8.0
MOVL C08823 V=8.0
MOVL C08824 V=8.0
MOVL C08825 V=8.0
MOVL C08826 V=8.0
MOVL C08827 V=8.0
MOVL C08828 V=8.0
MOVL C08829 V=8.0
MOVL C08830 V=8.0
MOVL C08831 V=8.0
MOVL C08832 V=8.0
MOVL C08833 V=8.0
MOVL C08834 V=8.0
MOVL C08835 V=8.0
MOVL C08836 V=8.0
MOVL C08837 V=8.0
MOVL C08838 V=8.0
MOVL C08839 V=8.0
MOVL C08840 V=8.0
MOVL C08841 V=8.0
MOVL C08842 V=8.0
MOVL C08843 V=8.0
MOVL C08844 V=8.0
MOVL C08845 V=8.0
MOVL C08846 V=8.0
MOVL C08847 V=8.0
MOVL C08848 V=8.0
MOVL C08849 V=8.0
MOVL C08850 V=8.0
MOVL C08851 V=8.0
MOVL C08852 V=8.0
MOVL C08853 V=8.0
MOVL C08854 V=8.0
MOVL C08855 V=8.0
MOVL C08856 V=8.0
MOVL C08857 V=8.0
MOVL C08858 V=8.0
MOVL C08859 V=8.0
MOVL C08860 V=8.0
MOVJ C08861 VJ=0.78
MOVL C08862 V=8.0
MOVL C08863 V=8.0
MOVL C08864 V=8.0
MOVL C08865 V=8.0
MOVL C08866 V=8.0
MOVL C08867 V=8.0
MOVL C08868 V=8.0
MOVL C08869 V=8.0
MOVL C08870 V=8.0
MOVL C08871 V=8.0
MOVL C08872 V=8.0
MOVL C08873 V=8.0
MOVL C08874 V=8.0
MOVL C08875 V=8.0
MOVL C08876 V=8.0
MOVL C08877 V=8.0
MOVL C08878 V=8.0
MOVL C08879 V=8.0
MOVL C08880 V=8.0
MOVL C08881 V=8.0
MOVL C08882 V=8.0
MOVL C08883 V=8.0
MOVL C08884 V=8.0
MOVL C08885 V=8.0
MOVL C08886 V=8.0
MOVL C08887 V=8.0
MOVL C08888 V=8.0
MOVL C08889 V=8.0
MOVL C08890 V=8.0
MOVL C08891 V=8.0
MOVL C08892 V=8.0
MOVL C08893 V=8.0
MOVL C08894 V=8.0
MOVL C08895 V=8.0
MOVL C08896 V=8.0
MOVL C08897 V=8.0
MOVL C08898 V=8.0
MOVL C08899 V=8.0
MOVL C08900 V=8.0
MOVL C08901 V=8.0
MOVL C08902 V=8.0
MOVL C08903 V=8.0
MOVL C08904 V=8.0
MOVL C08905 V=8.0
MOVL C08906 V=8.0
MOVL C08907 V=8.0
MOVL C08908 V=8.0
MOVL C08909 V=8.0
MOVL C08910 V=8.0
MOVL C08911 V=8.0
MOVL C08912 V=8.0
MOVL C08913 V=8.0
MOVL C08914 V=8.0
MOVL C08915 V=8.0
MOVL C08916 V=8.0
MOVL C08917 V=8.0
MOVL C08918 V=8.0
MOVL C08919 V=8.0
MOVL C08920 V=8.0
MOVL C08921 V=8.0
MOVL C08922 V=8.0
MOVJ C08923 VJ=0.78
MOVJ C08924 VJ=0.78
MOVL C08925 V=11.7
TIMER T=2.00
MOVL C08926 V=11.7
MOVJ C08927 VJ=0.78
MOVJ C08928 VJ=0.78
MOVL C08929 V=8.0
MOVL C08930 V=8.0
MOVJ C08931 VJ=0.78
MOVL C08932 V=8.0
MOVL C08933 V=8.0
MOVL C08934 V=8.0
MOVL C08935 V=8.0
MOVL C08936 V=8.0
MOVL C08937 V=8.0
MOVL C08938 V=8.0
MOVL C08939 V=8.0
MOVL C08940 V=8.0
MOVL C08941 V=8.0
MOVL C08942 V=8.0
MOVL C08943 V=8.0
MOVL C08944 V=8.0
MOVL C08945 V=8.0
MOVL C08946 V=8.0
MOVL C08947 V=8.0
MOVL C08948 V=8.0
MOVL C08949 V=8.0
MOVL C08950 V=8.0
MOVL C08951 V=8.0
MOVL C08952 V=8.0
MOVL C08953 V=8.0
MOVL C08954 V=8.0
MOVL C08955 V=8.0
MOVL C08956 V=8.0
MOVL C08957 V=8.0
MOVL C08958 V=8.0
MOVL C08959 V=8.0
MOVL C08960 V=8.0
MOVL C08961 V=8.0
MOVL C08962 V=8.0
MOVL C08963 V=8.0
MOVL C08964 V=8.0
MOVL C08965 V=8.0
MOVL C08966 V=8.0
MOVL C08967 V=8.0
MOVL C08968 V=8.0
MOVL C08969 V=8.0
MOVL C08970 V=8.0
MOVL C08971 V=8.0
MOVL C08972 V=8.0
MOVL C08973 V=8.0
MOVL C08974 V=8.0
MOVL C08975 V=8.0
MOVL C08976 V=8.0
MOVL C08977 V=8.0
MOVL C08978 V=8.0
MOVL C08979 V=8.0
MOVL C08980 V=8.0
MOVL C08981 V=8.0
MOVL C08982 V=8.0
MOVL C08983 V=8.0
MOVL C08984 V=8.0
MOVL C08985 V=8.0
MOVL C08986 V=8.0
MOVL C08987 V=8.0
MOVL C08988 V=8.0
MOVL C08989 V=8.0
MOVL C08990 V=8.0
MOVL C08991 V=8.0
MOVL C08992 V=8.0
MOVL C08993 V=8.0
MOVJ C08994 VJ=0.78
MOVL C08995 V=8.0
MOVL C08996 V=8.0
MOVL C08997 V=8.0
MOVL C08998 V=8.0
MOVL C08999 V=8.0
MOVL C09000 V=8.0
MOVL C09001 V=8.0
MOVL C09002 V=8.0
MOVL C09003 V=8.0
MOVL C09004 V=8.0
MOVL C09005 V=8.0
MOVL C09006 V=8.0
MOVL C09007 V=8.0
MOVL C09008 V=8.0
MOVL C09009 V=8.0
MOVL C09010 V=8.0
MOVL C09011 V=8.0
MOVL C09012 V=8.0
MOVL C09013 V=8.0
MOVL C09014 V=8.0
MOVL C09015 V=8.0
MOVL C09016 V=8.0
MOVL C09017 V=8.0
MOVL C09018 V=8.0
MOVL C09019 V=8.0
MOVL C09020 V=8.0
MOVL C09021 V=8.0
MOVL C09022 V=8.0
MOVL C09023 V=8.0
MOVL C09024 V=8.0
MOVL C09025 V=8.0
MOVL C09026 V=8.0
MOVL C09027 V=8.0
MOVL C09028 V=8.0
MOVL C09029 V=8.0
MOVL C09030 V=8.0
MOVL C09031 V=8.0
MOVL C09032 V=8.0
MOVL C09033 V=8.0
MOVL C09034 V=8.0
MOVL C09035 V=8.0
MOVL C09036 V=8.0
MOVL C09037 V=8.0
MOVL C09038 V=8.0
MOVL C09039 V=8.0
MOVL C09040 V=8.0
MOVL C09041 V=8.0
MOVL C09042 V=8.0
MOVL C09043 V=8.0
MOVL C09044 V=8.0
MOVL C09045 V=8.0
MOVL C09046 V=8.0
MOVL C09047 V=8.0
MOVL C09048 V=8.0
MOVL C09049 V=8.0
MOVL C09050 V=8.0
MOVL C09051 V=8.0
MOVL C09052 V=8.0
MOVL C09053 V=8.0
MOVL C09054 V=8.0
MOVL C09055 V=8.0
MOVL C09056 V=8.0
MOVJ C09057 VJ=0.78
MOVL C09058 V=8.0
MOVL C09059 V=8.0
MOVL C09060 V=8.0
MOVL C09061 V=8.0
MOVL C09062 V=8.0
MOVL C09063 V=8.0
MOVL C09064 V=8.0
MOVL C09065 V=8.0
MOVL C09066 V=8.0
MOVL C09067 V=8.0
MOVL C09068 V=8.0
MOVL C09069 V=8.0
MOVL C09070 V=8.0
MOVL C09071 V=8.0
MOVL C09072 V=8.0
MOVL C09073 V=8.0
MOVL C09074 V=8.0
MOVL C09075 V=8.0
MOVL C09076 V=8.0
MOVL C09077 V=8.0
MOVL C09078 V=8.0
MOVL C09079 V=8.0
MOVL C09080 V=8.0
MOVL C09081 V=8.0
MOVL C09082 V=8.0
MOVL C09083 V=8.0
MOVL C09084 V=8.0
MOVL C09085 V=8.0
MOVL C09086 V=8.0
MOVL C09087 V=8.0
MOVL C09088 V=8.0
MOVL C09089 V=8.0
MOVL C09090 V=8.0
MOVL C09091 V=8.0
MOVL C09092 V=8.0
MOVL C09093 V=8.0
MOVL C09094 V=8.0
MOVL C09095 V=8.0
MOVL C09096 V=8.0
MOVL C09097 V=8.0
MOVL C09098 V=8.0
MOVJ C09099 VJ=0.78
MOVJ C09100 VJ=0.78
MOVL C09101 V=11.7
TIMER T=2.00
MOVL C09102 V=11.7
MOVJ C09103 VJ=0.78
MOVJ C09104 VJ=0.78
MOVL C09105 V=8.0
MOVL C09106 V=8.0
MOVL C09107 V=8.0
MOVL C09108 V=8.0
MOVL C09109 V=8.0
MOVL C09110 V=8.0
MOVL C09111 V=8.0
MOVL C09112 V=8.0
MOVL C09113 V=8.0
MOVL C09114 V=8.0
MOVL C09115 V=8.0
MOVL C09116 V=8.0
MOVL C09117 V=8.0
MOVL C09118 V=8.0
MOVL C09119 V=8.0
MOVL C09120 V=8.0
MOVL C09121 V=8.0
MOVL C09122 V=8.0
MOVL C09123 V=8.0
MOVL C09124 V=8.0
MOVL C09125 V=8.0
MOVL C09126 V=8.0
MOVJ C09127 VJ=0.78
MOVL C09128 V=8.0
MOVL C09129 V=8.0
MOVL C09130 V=8.0
MOVL C09131 V=8.0
MOVL C09132 V=8.0
MOVL C09133 V=8.0
MOVL C09134 V=8.0
MOVL C09135 V=8.0
MOVL C09136 V=8.0
MOVL C09137 V=8.0
MOVL C09138 V=8.0
MOVL C09139 V=8.0
MOVL C09140 V=8.0
MOVL C09141 V=8.0
MOVL C09142 V=8.0
MOVL C09143 V=8.0
MOVL C09144 V=8.0
MOVL C09145 V=8.0
MOVL C09146 V=8.0
MOVL C09147 V=8.0
MOVL C09148 V=8.0
MOVL C09149 V=8.0
MOVL C09150 V=8.0
MOVL C09151 V=8.0
MOVL C09152 V=8.0
MOVL C09153 V=8.0
MOVL C09154 V=8.0
MOVL C09155 V=8.0
MOVL C09156 V=8.0
MOVL C09157 V=8.0
MOVL C09158 V=8.0
MOVL C09159 V=8.0
MOVL C09160 V=8.0
MOVL C09161 V=8.0
MOVL C09162 V=8.0
MOVL C09163 V=8.0
MOVL C09164 V=8.0
MOVL C09165 V=8.0
MOVL C09166 V=8.0
MOVL C09167 V=8.0
MOVL C09168 V=8.0
MOVL C09169 V=8.0
MOVL C09170 V=8.0
MOVL C09171 V=8.0
MOVL C09172 V=8.0
MOVL C09173 V=8.0
MOVL C09174 V=8.0
MOVL C09175 V=8.0
MOVL C09176 V=8.0
MOVL C09177 V=8.0
MOVL C09178 V=8.0
MOVL C09179 V=8.0
MOVL C09180 V=8.0
MOVL C09181 V=8.0
MOVL C09182 V=8.0
MOVL C09183 V=8.0
MOVL C09184 V=8.0
MOVL C09185 V=8.0
MOVL C09186 V=8.0
MOVL C09187 V=8.0
MOVL C09188 V=8.0
MOVL C09189 V=8.0
MOVJ C09190 VJ=0.78
MOVL C09191 V=8.0
MOVL C09192 V=8.0
MOVL C09193 V=8.0
MOVL C09194 V=8.0
MOVL C09195 V=8.0
MOVL C09196 V=8.0
MOVL C09197 V=8.0
MOVL C09198 V=8.0
MOVL C09199 V=8.0
MOVL C09200 V=8.0
MOVL C09201 V=8.0
MOVL C09202 V=8.0
MOVL C09203 V=8.0
MOVL C09204 V=8.0
MOVL C09205 V=8.0
MOVL C09206 V=8.0
MOVL C09207 V=8.0
MOVL C09208 V=8.0
MOVL C09209 V=8.0
MOVL C09210 V=8.0
MOVL C09211 V=8.0
MOVL C09212 V=8.0
MOVL C09213 V=8.0
MOVL C09214 V=8.0
MOVL C09215 V=8.0
MOVL C09216 V=8.0
MOVL C09217 V=8.0
MOVL C09218 V=8.0
MOVL C09219 V=8.0
MOVL C09220 V=8.0
MOVL C09221 V=8.0
MOVL C09222 V=8.0
MOVL C09223 V=8.0
MOVL C09224 V=8.0
MOVL C09225 V=8.0
MOVL C09226 V=8.0
MOVL C09227 V=8.0
MOVL C09228 V=8.0
MOVL C09229 V=8.0
MOVL C09230 V=8.0
MOVL C09231 V=8.0
MOVL C09232 V=8.0
MOVL C09233 V=8.0
MOVL C09234 V=8.0
MOVL C09235 V=8.0
MOVL C09236 V=8.0
MOVL C09237 V=8.0
MOVL C09238 V=8.0
MOVL C09239 V=8.0
MOVL C09240 V=8.0
MOVL C09241 V=8.0
MOVL C09242 V=8.0
MOVL C09243 V=8.0
MOVL C09244 V=8.0
MOVL C09245 V=8.0
MOVL C09246 V=8.0
MOVL C09247 V=8.0
MOVL C09248 V=8.0
MOVL C09249 V=8.0
MOVL C09250 V=8.0
MOVL C09251 V=8.0
MOVL C09252 V=8.0
MOVJ C09253 VJ=0.78
MOVL C09254 V=8.0
MOVL C09255 V=8.0
MOVL C09256 V=8.0
MOVL C09257 V=8.0
MOVL C09258 V=8.0
MOVL C09259 V=8.0
MOVL C09260 V=8.0
MOVL C09261 V=8.0
MOVL C09262 V=8.0
MOVL C09263 V=8.0
MOVL C09264 V=8.0
MOVL C09265 V=8.0
MOVL C09266 V=8.0
MOVL C09267 V=8.0
MOVL C09268 V=8.0
MOVL C09269 V=8.0
MOVL C09270 V=8.0
MOVL C09271 V=8.0
MOVL C09272 V=8.0
MOVL C09273 V=8.0
MOVL C09274 V=8.0
MOVJ C09275 VJ=0.78
MOVJ C09276 VJ=0.78
MOVL C09277 V=11.7
TIMER T=2.00
MOVL C09278 V=11.7
MOVJ C09279 VJ=0.78
MOVJ C09280 VJ=0.78
MOVL C09281 V=8.0
MOVL C09282 V=8.0
MOVL C09283 V=8.0
MOVL C09284 V=8.0
MOVL C09285 V=8.0
MOVL C09286 V=8.0
MOVL C09287 V=8.0
MOVL C09288 V=8.0
MOVL C09289 V=8.0
MOVL C09290 V=8.0
MOVL C09291 V=8.0
MOVL C09292 V=8.0
MOVL C09293 V=8.0
MOVL C09294 V=8.0
MOVL C09295 V=8.0
MOVL C09296 V=8.0
MOVL C09297 V=8.0
MOVL C09298 V=8.0
MOVL C09299 V=8.0
MOVL C09300 V=8.0
MOVL C09301 V=8.0
MOVL C09302 V=8.0
MOVL C09303 V=8.0
MOVL C09304 V=8.0
MOVL C09305 V=8.0
MOVL C09306 V=8.0
MOVL C09307 V=8.0
MOVL C09308 V=8.0
MOVL C09309 V=8.0
MOVL C09310 V=8.0
MOVL C09311 V=8.0
MOVL C09312 V=8.0
MOVL C09313 V=8.0
MOVL C09314 V=8.0
MOVL C09315 V=8.0
MOVL C09316 V=8.0
MOVL C09317 V=8.0
MOVL C09318 V=8.0
MOVL C09319 V=8.0
MOVL C09320 V=8.0
MOVL C09321 V=8.0
MOVL C09322 V=8.0
MOVJ C09323 VJ=0.78
MOVL C09324 V=8.0
MOVL C09325 V=8.0
MOVL C09326 V=8.0
MOVL C09327 V=8.0
MOVL C09328 V=8.0
MOVL C09329 V=8.0
MOVL C09330 V=8.0
MOVL C09331 V=8.0
MOVL C09332 V=8.0
MOVL C09333 V=8.0
MOVL C09334 V=8.0
MOVL C09335 V=8.0
MOVL C09336 V=8.0
MOVL C09337 V=8.0
MOVL C09338 V=8.0
MOVL C09339 V=8.0
MOVL C09340 V=8.0
MOVL C09341 V=8.0
MOVL C09342 V=8.0
MOVL C09343 V=8.0
MOVL C09344 V=8.0
MOVL C09345 V=8.0
MOVL C09346 V=8.0
MOVL C09347 V=8.0
MOVL C09348 V=8.0
MOVL C09349 V=8.0
MOVL C09350 V=8.0
MOVL C09351 V=8.0
MOVL C09352 V=8.0
MOVL C09353 V=8.0
MOVL C09354 V=8.0
MOVL C09355 V=8.0
MOVL C09356 V=8.0
MOVL C09357 V=8.0
MOVL C09358 V=8.0
MOVL C09359 V=8.0
MOVL C09360 V=8.0
MOVL C09361 V=8.0
MOVL C09362 V=8.0
MOVL C09363 V=8.0
MOVL C09364 V=8.0
MOVL C09365 V=8.0
MOVL C09366 V=8.0
MOVL C09367 V=8.0
MOVL C09368 V=8.0
MOVL C09369 V=8.0
MOVL C09370 V=8.0
MOVL C09371 V=8.0
MOVL C09372 V=8.0
MOVL C09373 V=8.0
MOVL C09374 V=8.0
MOVL C09375 V=8.0
MOVL C09376 V=8.0
MOVL C09377 V=8.0
MOVL C09378 V=8.0
MOVL C09379 V=8.0
MOVL C09380 V=8.0
MOVL C09381 V=8.0
MOVL C09382 V=8.0
MOVL C09383 V=8.0
MOVL C09384 V=8.0
MOVL C09385 V=8.0
MOVJ C09386 VJ=0.78
MOVL C09387 V=8.0
MOVL C09388 V=8.0
MOVL C09389 V=8.0
MOVL C09390 V=8.0
MOVL C09391 V=8.0
MOVL C09392 V=8.0
MOVL C09393 V=8.0
MOVL C09394 V=8.0
MOVL C09395 V=8.0
MOVL C09396 V=8.0
MOVL C09397 V=8.0
MOVL C09398 V=8.0
MOVL C09399 V=8.0
MOVL C09400 V=8.0
MOVL C09401 V=8.0
MOVL C09402 V=8.0
MOVL C09403 V=8.0
MOVL C09404 V=8.0
MOVL C09405 V=8.0
MOVL C09406 V=8.0
MOVL C09407 V=8.0
MOVL C09408 V=8.0
MOVL C09409 V=8.0
MOVL C09410 V=8.0
MOVL C09411 V=8.0
MOVL C09412 V=8.0
MOVL C09413 V=8.0
MOVL C09414 V=8.0
MOVL C09415 V=8.0
MOVL C09416 V=8.0
MOVL C09417 V=8.0
MOVL C09418 V=8.0
MOVL C09419 V=8.0
MOVL C09420 V=8.0
MOVL C09421 V=8.0
MOVL C09422 V=8.0
MOVL C09423 V=8.0
MOVL C09424 V=8.0
MOVL C09425 V=8.0
MOVL C09426 V=8.0
MOVL C09427 V=8.0
MOVL C09428 V=8.0
MOVL C09429 V=8.0
MOVL C09430 V=8.0
MOVL C09431 V=8.0
MOVL C09432 V=8.0
MOVL C09433 V=8.0
MOVL C09434 V=8.0
MOVL C09435 V=8.0
MOVL C09436 V=8.0
MOVL C09437 V=8.0
MOVL C09438 V=8.0
MOVL C09439 V=8.0
MOVL C09440 V=8.0
MOVL C09441 V=8.0
MOVL C09442 V=8.0
MOVL C09443 V=8.0
MOVL C09444 V=8.0
MOVL C09445 V=8.0
MOVL C09446 V=8.0
MOVL C09447 V=8.0
MOVJ C09448 VJ=0.78
MOVJ C09449 VJ=0.78
MOVL C09450 V=11.7
TIMER T=2.00
MOVL C09451 V=11.7
MOVJ C09452 VJ=0.78
MOVJ C09453 VJ=0.78
MOVL C09454 V=8.0
MOVL C09455 V=8.0
MOVJ C09456 VJ=0.78
MOVL C09457 V=8.0
MOVL C09458 V=8.0
MOVL C09459 V=8.0
MOVL C09460 V=8.0
MOVL C09461 V=8.0
MOVL C09462 V=8.0
MOVL C09463 V=8.0
MOVL C09464 V=8.0
MOVL C09465 V=8.0
MOVL C09466 V=8.0
MOVL C09467 V=8.0
MOVL C09468 V=8.0
MOVL C09469 V=8.0
MOVL C09470 V=8.0
MOVL C09471 V=8.0
MOVL C09472 V=8.0
MOVL C09473 V=8.0
MOVL C09474 V=8.0
MOVL C09475 V=8.0
MOVL C09476 V=8.0
MOVL C09477 V=8.0
MOVL C09478 V=8.0
MOVL C09479 V=8.0
MOVL C09480 V=8.0
MOVL C09481 V=8.0
MOVL C09482 V=8.0
MOVL C09483 V=8.0
MOVL C09484 V=8.0
MOVL C09485 V=8.0
MOVL C09486 V=8.0
MOVL C09487 V=8.0
MOVL C09488 V=8.0
MOVL C09489 V=8.0
MOVL C09490 V=8.0
MOVL C09491 V=8.0
MOVL C09492 V=8.0
MOVL C09493 V=8.0
MOVL C09494 V=8.0
MOVL C09495 V=8.0
MOVL C09496 V=8.0
MOVL C09497 V=8.0
MOVL C09498 V=8.0
MOVL C09499 V=8.0
MOVL C09500 V=8.0
MOVL C09501 V=8.0
MOVL C09502 V=8.0
MOVL C09503 V=8.0
MOVL C09504 V=8.0
MOVL C09505 V=8.0
MOVL C09506 V=8.0
MOVL C09507 V=8.0
MOVL C09508 V=8.0
MOVL C09509 V=8.0
MOVL C09510 V=8.0
MOVL C09511 V=8.0
MOVL C09512 V=8.0
MOVL C09513 V=8.0
MOVL C09514 V=8.0
MOVL C09515 V=8.0
MOVL C09516 V=8.0
MOVL C09517 V=8.0
MOVL C09518 V=8.0
MOVJ C09519 VJ=0.78
MOVL C09520 V=8.0
MOVL C09521 V=8.0
MOVL C09522 V=8.0
MOVL C09523 V=8.0
MOVL C09524 V=8.0
MOVL C09525 V=8.0
MOVL C09526 V=8.0
MOVL C09527 V=8.0
MOVL C09528 V=8.0
MOVL C09529 V=8.0
MOVL C09530 V=8.0
MOVL C09531 V=8.0
MOVL C09532 V=8.0
MOVL C09533 V=8.0
MOVL C09534 V=8.0
MOVL C09535 V=8.0
MOVL C09536 V=8.0
MOVL C09537 V=8.0
MOVL C09538 V=8.0
MOVL C09539 V=8.0
MOVL C09540 V=8.0
MOVL C09541 V=8.0
MOVL C09542 V=8.0
MOVL C09543 V=8.0
MOVL C09544 V=8.0
MOVL C09545 V=8.0
MOVL C09546 V=8.0
MOVL C09547 V=8.0
MOVL C09548 V=8.0
MOVL C09549 V=8.0
MOVL C09550 V=8.0
MOVL C09551 V=8.0
MOVL C09552 V=8.0
MOVL C09553 V=8.0
MOVL C09554 V=8.0
MOVL C09555 V=8.0
MOVL C09556 V=8.0
MOVL C09557 V=8.0
MOVL C09558 V=8.0
MOVL C09559 V=8.0
MOVL C09560 V=8.0
MOVL C09561 V=8.0
MOVL C09562 V=8.0
MOVL C09563 V=8.0
MOVL C09564 V=8.0
MOVL C09565 V=8.0
MOVL C09566 V=8.0
MOVL C09567 V=8.0
MOVL C09568 V=8.0
MOVL C09569 V=8.0
MOVL C09570 V=8.0
MOVL C09571 V=8.0
MOVL C09572 V=8.0
MOVL C09573 V=8.0
MOVL C09574 V=8.0
MOVL C09575 V=8.0
MOVL C09576 V=8.0
MOVL C09577 V=8.0
MOVL C09578 V=8.0
MOVL C09579 V=8.0
MOVL C09580 V=8.0
MOVL C09581 V=8.0
MOVJ C09582 VJ=0.78
MOVL C09583 V=8.0
MOVL C09584 V=8.0
MOVL C09585 V=8.0
MOVL C09586 V=8.0
MOVL C09587 V=8.0
MOVL C09588 V=8.0
MOVL C09589 V=8.0
MOVL C09590 V=8.0
MOVL C09591 V=8.0
MOVL C09592 V=8.0
MOVL C09593 V=8.0
MOVL C09594 V=8.0
MOVL C09595 V=8.0
MOVL C09596 V=8.0
MOVL C09597 V=8.0
MOVL C09598 V=8.0
MOVL C09599 V=8.0
MOVL C09600 V=8.0
MOVL C09601 V=8.0
MOVL C09602 V=8.0
MOVL C09603 V=8.0
MOVL C09604 V=8.0
MOVL C09605 V=8.0
MOVL C09606 V=8.0
MOVL C09607 V=8.0
MOVL C09608 V=8.0
MOVL C09609 V=8.0
MOVL C09610 V=8.0
MOVL C09611 V=8.0
MOVL C09612 V=8.0
MOVL C09613 V=8.0
MOVL C09614 V=8.0
MOVL C09615 V=8.0
MOVL C09616 V=8.0
MOVL C09617 V=8.0
MOVL C09618 V=8.0
MOVL C09619 V=8.0
MOVL C09620 V=8.0
MOVL C09621 V=8.0
MOVL C09622 V=8.0
MOVL C09623 V=8.0
MOVJ C09624 VJ=0.78
MOVJ C09625 VJ=0.78
MOVL C09626 V=11.7
TIMER T=2.00
MOVL C09627 V=11.7
MOVJ C09628 VJ=0.78
MOVJ C09629 VJ=0.78
MOVL C09630 V=8.0
MOVL C09631 V=8.0
MOVL C09632 V=8.0
MOVL C09633 V=8.0
MOVL C09634 V=8.0
MOVL C09635 V=8.0
MOVL C09636 V=8.0
MOVL C09637 V=8.0
MOVL C09638 V=8.0
MOVL C09639 V=8.0
MOVL C09640 V=8.0
MOVL C09641 V=8.0
MOVL C09642 V=8.0
MOVL C09643 V=8.0
MOVL C09644 V=8.0
MOVL C09645 V=8.0
MOVL C09646 V=8.0
MOVL C09647 V=8.0
MOVL C09648 V=8.0
MOVL C09649 V=8.0
MOVL C09650 V=8.0
MOVL C09651 V=8.0
MOVJ C09652 VJ=0.78
MOVL C09653 V=8.0
MOVL C09654 V=8.0
MOVL C09655 V=8.0
MOVL C09656 V=8.0
MOVL C09657 V=8.0
MOVL C09658 V=8.0
MOVL C09659 V=8.0
MOVL C09660 V=8.0
MOVL C09661 V=8.0
MOVL C09662 V=8.0
MOVL C09663 V=8.0
MOVL C09664 V=8.0
MOVL C09665 V=8.0
MOVL C09666 V=8.0
MOVL C09667 V=8.0
MOVL C09668 V=8.0
MOVL C09669 V=8.0
MOVL C09670 V=8.0
MOVL C09671 V=8.0
MOVL C09672 V=8.0
MOVL C09673 V=8.0
MOVL C09674 V=8.0
MOVL C09675 V=8.0
MOVL C09676 V=8.0
MOVL C09677 V=8.0
MOVL C09678 V=8.0
MOVL C09679 V=8.0
MOVL C09680 V=8.0
MOVL C09681 V=8.0
MOVL C09682 V=8.0
MOVL C09683 V=8.0
MOVL C09684 V=8.0
MOVL C09685 V=8.0
MOVL C09686 V=8.0
MOVL C09687 V=8.0
MOVL C09688 V=8.0
MOVL C09689 V=8.0
MOVL C09690 V=8.0
MOVL C09691 V=8.0
MOVL C09692 V=8.0
MOVL C09693 V=8.0
MOVL C09694 V=8.0
MOVL C09695 V=8.0
MOVL C09696 V=8.0
MOVL C09697 V=8.0
MOVL C09698 V=8.0
MOVL C09699 V=8.0
MOVL C09700 V=8.0
MOVL C09701 V=8.0
MOVL C09702 V=8.0
MOVL C09703 V=8.0
MOVL C09704 V=8.0
MOVL C09705 V=8.0
MOVL C09706 V=8.0
MOVL C09707 V=8.0
MOVL C09708 V=8.0
MOVL C09709 V=8.0
MOVL C09710 V=8.0
MOVL C09711 V=8.0
MOVL C09712 V=8.0
MOVL C09713 V=8.0
MOVL C09714 V=8.0
MOVJ C09715 VJ=0.78
MOVL C09716 V=8.0
MOVL C09717 V=8.0
MOVL C09718 V=8.0
MOVL C09719 V=8.0
MOVL C09720 V=8.0
MOVL C09721 V=8.0
MOVL C09722 V=8.0
MOVL C09723 V=8.0
MOVL C09724 V=8.0
MOVL C09725 V=8.0
MOVL C09726 V=8.0
MOVL C09727 V=8.0
MOVL C09728 V=8.0
MOVL C09729 V=8.0
MOVL C09730 V=8.0
MOVL C09731 V=8.0
MOVL C09732 V=8.0
MOVL C09733 V=8.0
MOVL C09734 V=8.0
MOVL C09735 V=8.0
MOVL C09736 V=8.0
MOVL C09737 V=8.0
MOVL C09738 V=8.0
MOVL C09739 V=8.0
MOVL C09740 V=8.0
MOVL C09741 V=8.0
MOVL C09742 V=8.0
MOVL C09743 V=8.0
MOVL C09744 V=8.0
MOVL C09745 V=8.0
MOVL C09746 V=8.0
MOVL C09747 V=8.0
MOVL C09748 V=8.0
MOVL C09749 V=8.0
MOVL C09750 V=8.0
MOVL C09751 V=8.0
MOVL C09752 V=8.0
MOVL C09753 V=8.0
MOVL C09754 V=8.0
MOVL C09755 V=8.0
MOVL C09756 V=8.0
MOVL C09757 V=8.0
MOVL C09758 V=8.0
MOVL C09759 V=8.0
MOVL C09760 V=8.0
MOVL C09761 V=8.0
MOVL C09762 V=8.0
MOVL C09763 V=8.0
MOVL C09764 V=8.0
MOVL C09765 V=8.0
MOVL C09766 V=8.0
MOVL C09767 V=8.0
MOVL C09768 V=8.0
MOVL C09769 V=8.0
MOVL C09770 V=8.0
MOVL C09771 V=8.0
MOVL C09772 V=8.0
MOVL C09773 V=8.0
MOVL C09774 V=8.0
MOVL C09775 V=8.0
MOVL C09776 V=8.0
MOVL C09777 V=8.0
MOVJ C09778 VJ=0.78
MOVL C09779 V=8.0
MOVL C09780 V=8.0
MOVL C09781 V=8.0
MOVL C09782 V=8.0
MOVL C09783 V=8.0
MOVL C09784 V=8.0
MOVL C09785 V=8.0
MOVL C09786 V=8.0
MOVL C09787 V=8.0
MOVL C09788 V=8.0
MOVL C09789 V=8.0
MOVL C09790 V=8.0
MOVL C09791 V=8.0
MOVL C09792 V=8.0
MOVL C09793 V=8.0
MOVL C09794 V=8.0
MOVL C09795 V=8.0
MOVL C09796 V=8.0
MOVL C09797 V=8.0
MOVL C09798 V=8.0
MOVL C09799 V=8.0
MOVJ C09800 VJ=0.78
MOVJ C09801 VJ=0.78
MOVL C09802 V=11.7
TIMER T=2.00
MOVL C09803 V=11.7
MOVJ C09804 VJ=0.78
MOVJ C09805 VJ=0.78
MOVL C09806 V=8.0
MOVL C09807 V=8.0
MOVL C09808 V=8.0
MOVL C09809 V=8.0
MOVL C09810 V=8.0
MOVL C09811 V=8.0
MOVL C09812 V=8.0
MOVL C09813 V=8.0
MOVL C09814 V=8.0
MOVL C09815 V=8.0
MOVL C09816 V=8.0
MOVL C09817 V=8.0
MOVL C09818 V=8.0
MOVL C09819 V=8.0
MOVL C09820 V=8.0
MOVL C09821 V=8.0
MOVL C09822 V=8.0
MOVL C09823 V=8.0
MOVL C09824 V=8.0
MOVL C09825 V=8.0
MOVL C09826 V=8.0
MOVL C09827 V=8.0
MOVL C09828 V=8.0
MOVL C09829 V=8.0
MOVL C09830 V=8.0
MOVL C09831 V=8.0
MOVL C09832 V=8.0
MOVL C09833 V=8.0
MOVL C09834 V=8.0
MOVL C09835 V=8.0
MOVL C09836 V=8.0
MOVL C09837 V=8.0
MOVL C09838 V=8.0
MOVL C09839 V=8.0
MOVL C09840 V=8.0
MOVL C09841 V=8.0
MOVL C09842 V=8.0
MOVL C09843 V=8.0
MOVL C09844 V=8.0
MOVL C09845 V=8.0
MOVL C09846 V=8.0
MOVL C09847 V=8.0
END
